  PROC DrawPart154()
    MoveL Offs(pOrigin,203.09,148.13,0.00),v40,z0,tPen\WObj:=wPaper;
    MoveL Offs(pOrigin,201.29,146.33,0.00),v40,z0,tPen\WObj:=wPaper;
    MoveL Offs(pOrigin,200.72,146.00,0.00),v40,z0,tPen\WObj:=wPaper;
    MoveL Offs(pOrigin,205.53,141.19,0.00),v40,z0,tPen\WObj:=wPaper;
    MoveL Offs(pOrigin,205.02,141.09,0.00),v40,z0,tPen\WObj:=wPaper;
    MoveL Offs(pOrigin,203.22,139.29,0.00),v40,z0,tPen\WObj:=wPaper;
    MoveL Offs(pOrigin,203.68,139.61,0.00),v40,z0,tPen\WObj:=wPaper;
    MoveL Offs(pOrigin,204.95,139.61,0.00),v40,z0,tPen\WObj:=wPaper;
    MoveL Offs(pOrigin,205.31,139.90,0.00),v40,z0,tPen\WObj:=wPaper;
    MoveL Offs(pOrigin,203.51,138.09,0.00),v40,z0,tPen\WObj:=wPaper;
    MoveL Offs(pOrigin,202.84,137.91,0.00),v40,z0,tPen\WObj:=wPaper;
    MoveL Offs(pOrigin,207.80,132.95,0.00),v40,z0,tPen\WObj:=wPaper;
    MoveL Offs(pOrigin,207.24,132.86,0.00),v40,z0,tPen\WObj:=wPaper;
    MoveL Offs(pOrigin,205.44,131.06,0.00),v40,z0,tPen\WObj:=wPaper;
    MoveL Offs(pOrigin,206.01,131.16,0.00),v40,z0,tPen\WObj:=wPaper;
    MoveL Offs(pOrigin,207.29,131.16,0.00),v40,z0,tPen\WObj:=wPaper;
    MoveL Offs(pOrigin,207.69,131.82,0.00),v40,z0,tPen\WObj:=wPaper;
    MoveL Offs(pOrigin,205.73,129.86,0.00),v40,z0,tPen\WObj:=wPaper;
    MoveL Offs(pOrigin,206.23,130.10,0.00),v40,z0,tPen\WObj:=wPaper;
    MoveL Offs(pOrigin,207.71,130.10,0.00),v40,z0,tPen\WObj:=wPaper;
    MoveL Offs(pOrigin,208.13,130.77,0.00),v40,z0,tPen\WObj:=wPaper;
    MoveL Offs(pOrigin,205.88,128.51,0.00),v40,z0,tPen\WObj:=wPaper;
    MoveL Offs(pOrigin,206.44,129.05,0.00),v40,z0,tPen\WObj:=wPaper;
    MoveL Offs(pOrigin,207.92,129.05,0.00),v40,z0,tPen\WObj:=wPaper;
    MoveL Offs(pOrigin,208.28,129.42,0.00),v40,z0,tPen\WObj:=wPaper;
    MoveL Offs(pOrigin,206.02,127.17,0.00),v40,z0,tPen\WObj:=wPaper;
    MoveL Offs(pOrigin,206.86,126.94,0.00),v40,z0,tPen\WObj:=wPaper;
    MoveL Offs(pOrigin,208.56,126.94,0.00),v40,z0,tPen\WObj:=wPaper;
    MoveL Offs(pOrigin,209.02,127.18,0.00),v40,z0,tPen\WObj:=wPaper;
    MoveL Offs(pOrigin,206.47,124.62,0.00),v40,z0,tPen\WObj:=wPaper;
    MoveL Offs(pOrigin,206.03,124.27,0.00),v40,z0,tPen\WObj:=wPaper;
    MoveL Offs(pOrigin,212.04,118.26,0.00),v40,z0,tPen\WObj:=wPaper;
    MoveL Offs(pOrigin,211.69,117.90,0.00),v40,z0,tPen\WObj:=wPaper;
    MoveL Offs(pOrigin,208.23,114.44,0.00),v40,z0,tPen\WObj:=wPaper;
    MoveL Offs(pOrigin,207.56,113.77,0.00),v40,z0,tPen\WObj:=wPaper;
    MoveL Offs(pOrigin,215.37,105.96,0.00),v40,z0,tPen\WObj:=wPaper;
    MoveL Offs(pOrigin,214.65,105.92,0.00),v40,z0,tPen\WObj:=wPaper;
    MoveL Offs(pOrigin,212.99,104.27,0.00),v40,z0,tPen\WObj:=wPaper;
    MoveL Offs(pOrigin,213.24,104.76,0.00),v40,z0,tPen\WObj:=wPaper;
    MoveL Offs(pOrigin,214.51,104.76,0.00),v40,z0,tPen\WObj:=wPaper;
    MoveL Offs(pOrigin,215.09,104.87,0.00),v40,z0,tPen\WObj:=wPaper;
    MoveL Offs(pOrigin,213.14,102.92,0.00),v40,z0,tPen\WObj:=wPaper;
    MoveL Offs(pOrigin,212.53,102.82,0.00),v40,z0,tPen\WObj:=wPaper;
    MoveL Offs(pOrigin,216.89,98.47,0.00),v40,z0,tPen\WObj:=wPaper;
    MoveL Offs(pOrigin,216.42,98.74,0.00),v40,z0,tPen\WObj:=wPaper;
    MoveL Offs(pOrigin,214.47,96.78,0.00),v40,z0,tPen\WObj:=wPaper;
    MoveL Offs(pOrigin,214.72,97.37,0.00),v40,z0,tPen\WObj:=wPaper;
    MoveL Offs(pOrigin,216.00,97.37,0.00),v40,z0,tPen\WObj:=wPaper;
    MoveL Offs(pOrigin,216.57,97.39,0.00),v40,z0,tPen\WObj:=wPaper;
    MoveL Offs(pOrigin,214.47,95.29,0.00),v40,z0,tPen\WObj:=wPaper;
    MoveL Offs(pOrigin,214.06,95.33,0.00),v40,z0,tPen\WObj:=wPaper;
    MoveL Offs(pOrigin,217.96,91.42,0.00),v40,z0,tPen\WObj:=wPaper;
    MoveL Offs(pOrigin,217.45,90.80,0.00),v40,z0,tPen\WObj:=wPaper;
    MoveL Offs(pOrigin,215.49,88.85,0.00),v40,z0,tPen\WObj:=wPaper;
    MoveL Offs(pOrigin,216.00,88.92,0.00),v40,z0,tPen\WObj:=wPaper;
    MoveL Offs(pOrigin,217.28,88.92,0.00),v40,z0,tPen\WObj:=wPaper;
    MoveL Offs(pOrigin,217.59,89.45,0.00),v40,z0,tPen\WObj:=wPaper;
    MoveL Offs(pOrigin,215.49,87.35,0.00),v40,z0,tPen\WObj:=wPaper;
    MoveL Offs(pOrigin,215.13,86.79,0.00),v40,z0,tPen\WObj:=wPaper;
    MoveL Offs(pOrigin,218.74,83.18,0.00),v40,z0,tPen\WObj:=wPaper;
    MoveL Offs(pOrigin,218.17,82.56,0.00),v40,z0,tPen\WObj:=wPaper;
    MoveL Offs(pOrigin,216.07,80.46,0.00),v40,z0,tPen\WObj:=wPaper;
    MoveL Offs(pOrigin,216.64,80.47,0.00),v40,z0,tPen\WObj:=wPaper;
    MoveL Offs(pOrigin,217.91,80.47,0.00),v40,z0,tPen\WObj:=wPaper;
    MoveL Offs(pOrigin,218.17,81.07,0.00),v40,z0,tPen\WObj:=wPaper;
    MoveL Offs(pOrigin,216.06,78.96,0.00),v40,z0,tPen\WObj:=wPaper;
    MoveL Offs(pOrigin,215.60,78.85,0.00),v40,z0,tPen\WObj:=wPaper;
    MoveL Offs(pOrigin,218.91,75.54,0.00),v40,z0,tPen\WObj:=wPaper;
    MoveL Offs(pOrigin,218.45,75.37,0.00),v40,z0,tPen\WObj:=wPaper;
    MoveL Offs(pOrigin,216.04,72.97,0.00),v40,z0,tPen\WObj:=wPaper;
    MoveL Offs(pOrigin,215.62,72.85,0.00),v40,z0,tPen\WObj:=wPaper;
    MoveL Offs(pOrigin,218.93,69.55,0.00),v40,z0,tPen\WObj:=wPaper;
    MoveL Offs(pOrigin,218.58,69.53,0.00),v40,z0,tPen\WObj:=wPaper;
    MoveL Offs(pOrigin,211.67,62.62,0.00),v40,z0,tPen\WObj:=wPaper;
    MoveL Offs(pOrigin,211.54,62.80,0.00),v40,z0,tPen\WObj:=wPaper;
    MoveL Offs(pOrigin,211.11,63.22,0.00),v40,z0,tPen\WObj:=wPaper;
    MoveL Offs(pOrigin,211.54,62.80,0.00),v40,fine,tPen\WObj:=wPaper;
    MoveL Offs(pOrigin,211.54,62.80,6.00),v60,z5,tPen\WObj:=wPaper;
    MoveL Offs(pOrigin,212.26,61.72,6.00),vTravel,z5,tPen\WObj:=wPaper;
    MoveL Offs(pOrigin,212.26,61.72,0.00),v60,z0,tPen\WObj:=wPaper;
    MoveL Offs(pOrigin,218.28,67.73,0.00),v40,z0,tPen\WObj:=wPaper;
    MoveL Offs(pOrigin,217.91,67.80,0.00),v40,z0,tPen\WObj:=wPaper;
    MoveL Offs(pOrigin,214.51,67.80,0.00),v40,z0,tPen\WObj:=wPaper;
    MoveL Offs(pOrigin,214.08,68.02,0.00),v40,z0,tPen\WObj:=wPaper;
    MoveL Offs(pOrigin,218.59,72.53,0.00),v40,z0,tPen\WObj:=wPaper;
    MoveL Offs(pOrigin,218.92,72.55,0.00),v40,z0,tPen\WObj:=wPaper;
    MoveL Offs(pOrigin,215.61,75.85,0.00),v40,z0,tPen\WObj:=wPaper;
    MoveL Offs(pOrigin,216.05,75.97,0.00),v40,z0,tPen\WObj:=wPaper;
    MoveL Offs(pOrigin,218.46,78.37,0.00),v40,z0,tPen\WObj:=wPaper;
    MoveL Offs(pOrigin,218.90,78.54,0.00),v40,z0,tPen\WObj:=wPaper;
    MoveL Offs(pOrigin,215.44,81.99,0.00),v40,z0,tPen\WObj:=wPaper;
    MoveL Offs(pOrigin,215.92,81.81,0.00),v40,z0,tPen\WObj:=wPaper;
    MoveL Offs(pOrigin,218.03,83.91,0.00),v40,z0,tPen\WObj:=wPaper;
    MoveL Offs(pOrigin,217.70,83.64,0.00),v40,z0,tPen\WObj:=wPaper;
    MoveL Offs(pOrigin,216.42,83.64,0.00),v40,z0,tPen\WObj:=wPaper;
    MoveL Offs(pOrigin,215.93,83.31,0.00),v40,z0,tPen\WObj:=wPaper;
    MoveL Offs(pOrigin,218.03,85.41,0.00),v40,z0,tPen\WObj:=wPaper;
    MoveL Offs(pOrigin,217.49,85.75,0.00),v40,z0,tPen\WObj:=wPaper;
    MoveL Offs(pOrigin,216.21,85.75,0.00),v40,z0,tPen\WObj:=wPaper;
    MoveL Offs(pOrigin,215.63,86.00,0.00),v40,z0,tPen\WObj:=wPaper;
    MoveL Offs(pOrigin,217.89,88.26,0.00),v40,z0,tPen\WObj:=wPaper;
    MoveL Offs(pOrigin,218.27,88.13,0.00),v40,z0,tPen\WObj:=wPaper;
    MoveL Offs(pOrigin,214.67,91.73,0.00),v40,z0,tPen\WObj:=wPaper;
    MoveL Offs(pOrigin,215.05,91.39,0.00),v40,z0,tPen\WObj:=wPaper;
    MoveL Offs(pOrigin,217.16,93.50,0.00),v40,z0,tPen\WObj:=wPaper;
    MoveL Offs(pOrigin,217.66,93.22,0.00),v40,z0,tPen\WObj:=wPaper;
    MoveL Offs(pOrigin,213.75,97.13,0.00),v40,z0,tPen\WObj:=wPaper;
    MoveL Offs(pOrigin,214.02,97.83,0.00),v40,z0,tPen\WObj:=wPaper;
    MoveL Offs(pOrigin,216.13,99.93,0.00),v40,z0,tPen\WObj:=wPaper;
    MoveL Offs(pOrigin,216.44,100.42,0.00),v40,z0,tPen\WObj:=wPaper;
    MoveL Offs(pOrigin,212.08,104.77,0.00),v40,z0,tPen\WObj:=wPaper;
    MoveL Offs(pOrigin,212.55,105.32,0.00),v40,z0,tPen\WObj:=wPaper;
    MoveL Offs(pOrigin,214.50,107.27,0.00),v40,z0,tPen\WObj:=wPaper;
    MoveL Offs(pOrigin,214.09,106.87,0.00),v40,z0,tPen\WObj:=wPaper;
    MoveL Offs(pOrigin,212.81,106.87,0.00),v40,z0,tPen\WObj:=wPaper;
    MoveL Offs(pOrigin,212.25,106.51,0.00),v40,z0,tPen\WObj:=wPaper;
    MoveL Offs(pOrigin,214.36,108.62,0.00),v40,z0,tPen\WObj:=wPaper;
    MoveL Offs(pOrigin,214.61,108.21,0.00),v40,z0,tPen\WObj:=wPaper;
    MoveL Offs(pOrigin,207.40,115.42,0.00),v40,z0,tPen\WObj:=wPaper;
    MoveL Offs(pOrigin,207.94,115.64,0.00),v40,z0,tPen\WObj:=wPaper;
  ENDPROC

  PROC DrawPart155()
    MoveL Offs(pOrigin,211.24,118.94,0.00),v40,z0,tPen\WObj:=wPaper;
    MoveL Offs(pOrigin,210.90,118.49,0.00),v40,z0,tPen\WObj:=wPaper;
    MoveL Offs(pOrigin,209.41,118.49,0.00),v40,z0,tPen\WObj:=wPaper;
    MoveL Offs(pOrigin,209.84,117.43,0.00),v40,z0,tPen\WObj:=wPaper;
    MoveL Offs(pOrigin,211.32,117.43,0.00),v40,z0,tPen\WObj:=wPaper;
    MoveL Offs(pOrigin,211.98,116.70,0.00),v40,z0,tPen\WObj:=wPaper;
    MoveL Offs(pOrigin,208.53,113.24,0.00),v40,fine,tPen\WObj:=wPaper;
    MoveL Offs(pOrigin,208.53,113.24,6.00),v60,z5,tPen\WObj:=wPaper;
    MoveL Offs(pOrigin,207.86,111.98,6.00),vTravel,z5,tPen\WObj:=wPaper;
    MoveL Offs(pOrigin,207.86,111.98,0.00),v60,z0,tPen\WObj:=wPaper;
    MoveL Offs(pOrigin,210.27,109.57,0.00),v40,z0,tPen\WObj:=wPaper;
    MoveL Offs(pOrigin,211.02,108.82,0.00),v40,z0,tPen\WObj:=wPaper;
    MoveL Offs(pOrigin,215.83,104.01,0.00),v40,z0,tPen\WObj:=wPaper;
    MoveL Offs(pOrigin,215.39,103.68,0.00),v40,z0,tPen\WObj:=wPaper;
    MoveL Offs(pOrigin,213.44,101.72,0.00),v40,z0,tPen\WObj:=wPaper;
    MoveL Offs(pOrigin,214.09,101.59,0.00),v40,z0,tPen\WObj:=wPaper;
    MoveL Offs(pOrigin,215.15,101.59,0.00),v40,z0,tPen\WObj:=wPaper;
    MoveL Offs(pOrigin,215.83,101.13,0.00),v40,z0,tPen\WObj:=wPaper;
    MoveL Offs(pOrigin,213.88,99.18,0.00),v40,z0,tPen\WObj:=wPaper;
    MoveL Offs(pOrigin,213.45,98.93,0.00),v40,z0,tPen\WObj:=wPaper;
    MoveL Offs(pOrigin,217.50,94.87,0.00),v40,z0,tPen\WObj:=wPaper;
    MoveL Offs(pOrigin,217.01,94.84,0.00),v40,z0,tPen\WObj:=wPaper;
    MoveL Offs(pOrigin,214.76,92.59,0.00),v40,z0,tPen\WObj:=wPaper;
    MoveL Offs(pOrigin,215.58,92.09,0.00),v40,z0,tPen\WObj:=wPaper;
    MoveL Offs(pOrigin,216.85,92.09,0.00),v40,z0,tPen\WObj:=wPaper;
    MoveL Offs(pOrigin,217.15,92.00,0.00),v40,z0,tPen\WObj:=wPaper;
    MoveL Offs(pOrigin,215.20,90.04,0.00),v40,z0,tPen\WObj:=wPaper;
    MoveL Offs(pOrigin,214.82,90.08,0.00),v40,z0,tPen\WObj:=wPaper;
    MoveL Offs(pOrigin,218.58,86.33,0.00),v40,z0,tPen\WObj:=wPaper;
    MoveL Offs(pOrigin,217.88,86.76,0.00),v40,z0,tPen\WObj:=wPaper;
    MoveL Offs(pOrigin,215.63,84.50,0.00),v40,z0,tPen\WObj:=wPaper;
    MoveL Offs(pOrigin,215.28,85.14,0.00),v40,z0,tPen\WObj:=wPaper;
    MoveL Offs(pOrigin,218.74,81.68,0.00),v40,z0,tPen\WObj:=wPaper;
    MoveL Offs(pOrigin,217.91,81.53,0.00),v40,z0,tPen\WObj:=wPaper;
    MoveL Offs(pOrigin,216.64,81.53,0.00),v40,z0,tPen\WObj:=wPaper;
    MoveL Offs(pOrigin,216.64,82.58,0.00),v40,z0,tPen\WObj:=wPaper;
    MoveL Offs(pOrigin,217.70,82.58,0.00),v40,fine,tPen\WObj:=wPaper;
    MoveL Offs(pOrigin,217.70,82.58,6.00),v60,z5,tPen\WObj:=wPaper;
    MoveL Offs(pOrigin,217.49,84.70,6.00),vTravel,z5,tPen\WObj:=wPaper;
    MoveL Offs(pOrigin,217.49,84.70,0.00),v60,z0,tPen\WObj:=wPaper;
    MoveL Offs(pOrigin,216.42,84.70,0.00),v40,fine,tPen\WObj:=wPaper;
    MoveL Offs(pOrigin,216.42,84.70,6.00),v60,z5,tPen\WObj:=wPaper;
    MoveL Offs(pOrigin,215.29,83.64,6.00),vTravel,z5,tPen\WObj:=wPaper;
    MoveL Offs(pOrigin,215.29,83.64,0.00),v60,z0,tPen\WObj:=wPaper;
    MoveL Offs(pOrigin,219.05,79.88,0.00),v40,z0,tPen\WObj:=wPaper;
    MoveL Offs(pOrigin,218.46,79.87,0.00),v40,z0,tPen\WObj:=wPaper;
    MoveL Offs(pOrigin,216.06,77.46,0.00),v40,z0,tPen\WObj:=wPaper;
    MoveL Offs(pOrigin,215.61,77.35,0.00),v40,z0,tPen\WObj:=wPaper;
    MoveL Offs(pOrigin,218.91,74.04,0.00),v40,z0,tPen\WObj:=wPaper;
    MoveL Offs(pOrigin,218.59,74.03,0.00),v40,z0,tPen\WObj:=wPaper;
    MoveL Offs(pOrigin,213.79,69.22,0.00),v40,z0,tPen\WObj:=wPaper;
    MoveL Offs(pOrigin,214.09,69.91,0.00),v40,z0,tPen\WObj:=wPaper;
    MoveL Offs(pOrigin,217.91,69.91,0.00),v40,z0,tPen\WObj:=wPaper;
    MoveL Offs(pOrigin,217.91,68.86,0.00),v40,z0,tPen\WObj:=wPaper;
    MoveL Offs(pOrigin,214.51,68.86,0.00),v40,z0,tPen\WObj:=wPaper;
    MoveL Offs(pOrigin,215.44,68.54,0.00),v40,z0,tPen\WObj:=wPaper;
    MoveL Offs(pOrigin,215.44,59.82,0.00),v40,fine,tPen\WObj:=wPaper;
    MoveL Offs(pOrigin,215.44,59.82,6.00),v60,z5,tPen\WObj:=wPaper;
    MoveL Offs(pOrigin,213.76,60.23,6.00),vTravel,z5,tPen\WObj:=wPaper;
    MoveL Offs(pOrigin,213.76,60.23,0.00),v60,z0,tPen\WObj:=wPaper;
    MoveL Offs(pOrigin,218.12,64.59,0.00),v40,z0,tPen\WObj:=wPaper;
    MoveL Offs(pOrigin,217.49,64.63,0.00),v40,z0,tPen\WObj:=wPaper;
    MoveL Offs(pOrigin,214.51,64.63,0.00),v40,z0,tPen\WObj:=wPaper;
    MoveL Offs(pOrigin,214.51,65.69,0.00),v40,z0,tPen\WObj:=wPaper;
    MoveL Offs(pOrigin,217.70,65.69,0.00),v40,z0,tPen\WObj:=wPaper;
    MoveL Offs(pOrigin,217.70,66.74,0.00),v40,z0,tPen\WObj:=wPaper;
    MoveL Offs(pOrigin,214.51,66.74,0.00),v40,z0,tPen\WObj:=wPaper;
    MoveL Offs(pOrigin,214.08,66.52,0.00),v40,z0,tPen\WObj:=wPaper;
    MoveL Offs(pOrigin,218.59,71.03,0.00),v40,z0,tPen\WObj:=wPaper;
    MoveL Offs(pOrigin,218.92,71.05,0.00),v40,z0,tPen\WObj:=wPaper;
    MoveL Offs(pOrigin,215.62,74.35,0.00),v40,z0,tPen\WObj:=wPaper;
    MoveL Offs(pOrigin,216.05,74.47,0.00),v40,z0,tPen\WObj:=wPaper;
    MoveL Offs(pOrigin,218.45,76.87,0.00),v40,z0,tPen\WObj:=wPaper;
    MoveL Offs(pOrigin,218.90,77.04,0.00),v40,z0,tPen\WObj:=wPaper;
    MoveL Offs(pOrigin,215.45,80.50,0.00),v40,fine,tPen\WObj:=wPaper;
    MoveL Offs(pOrigin,215.45,80.50,6.00),v60,z5,tPen\WObj:=wPaper;
    MoveL Offs(pOrigin,216.64,79.42,6.00),vTravel,z5,tPen\WObj:=wPaper;
    MoveL Offs(pOrigin,216.64,79.42,0.00),v60,z0,tPen\WObj:=wPaper;
    MoveL Offs(pOrigin,217.91,79.42,0.00),v40,z0,tPen\WObj:=wPaper;
    MoveL Offs(pOrigin,217.91,78.36,0.00),v40,z0,tPen\WObj:=wPaper;
    MoveL Offs(pOrigin,216.85,78.36,0.00),v40,z0,tPen\WObj:=wPaper;
    MoveL Offs(pOrigin,216.85,77.30,0.00),v40,z0,tPen\WObj:=wPaper;
    MoveL Offs(pOrigin,217.91,77.30,0.00),v40,z0,tPen\WObj:=wPaper;
    MoveL Offs(pOrigin,217.91,76.25,0.00),v40,z0,tPen\WObj:=wPaper;
    MoveL Offs(pOrigin,216.85,76.25,0.00),v40,z0,tPen\WObj:=wPaper;
    MoveL Offs(pOrigin,216.85,75.19,0.00),v40,z0,tPen\WObj:=wPaper;
    MoveL Offs(pOrigin,217.91,75.19,0.00),v40,z0,tPen\WObj:=wPaper;
    MoveL Offs(pOrigin,217.91,74.14,0.00),v40,z0,tPen\WObj:=wPaper;
    MoveL Offs(pOrigin,216.85,74.14,0.00),v40,z0,tPen\WObj:=wPaper;
    MoveL Offs(pOrigin,216.85,73.08,0.00),v40,z0,tPen\WObj:=wPaper;
    MoveL Offs(pOrigin,217.91,73.08,0.00),v40,z0,tPen\WObj:=wPaper;
    MoveL Offs(pOrigin,217.91,72.02,0.00),v40,z0,tPen\WObj:=wPaper;
    MoveL Offs(pOrigin,216.85,72.02,0.00),v40,z0,tPen\WObj:=wPaper;
    MoveL Offs(pOrigin,216.85,70.97,0.00),v40,z0,tPen\WObj:=wPaper;
    MoveL Offs(pOrigin,217.91,70.97,0.00),v40,fine,tPen\WObj:=wPaper;
    MoveL Offs(pOrigin,217.91,70.97,6.00),v60,z5,tPen\WObj:=wPaper;
    MoveL Offs(pOrigin,218.63,68.35,6.00),vTravel,z5,tPen\WObj:=wPaper;
    MoveL Offs(pOrigin,218.63,68.35,0.00),v60,z0,tPen\WObj:=wPaper;
    MoveL Offs(pOrigin,212.77,74.21,0.00),v40,z0,tPen\WObj:=wPaper;
    MoveL Offs(pOrigin,212.60,74.01,0.00),v40,z0,tPen\WObj:=wPaper;
    MoveL Offs(pOrigin,210.95,72.36,0.00),v40,z0,tPen\WObj:=wPaper;
    MoveL Offs(pOrigin,210.26,73.08,0.00),v40,z0,tPen\WObj:=wPaper;
    MoveL Offs(pOrigin,212.60,73.08,0.00),v40,z0,tPen\WObj:=wPaper;
    MoveL Offs(pOrigin,213.24,73.00,0.00),v40,z0,tPen\WObj:=wPaper;
    MoveL Offs(pOrigin,213.52,72.86,0.00),v40,z0,tPen\WObj:=wPaper;
    MoveL Offs(pOrigin,210.90,74.35,0.00),v40,z0,tPen\WObj:=wPaper;
    MoveL Offs(pOrigin,206.86,75.55,0.00),v40,z0,tPen\WObj:=wPaper;
    MoveL Offs(pOrigin,204.10,75.97,0.00),v40,z0,tPen\WObj:=wPaper;
    MoveL Offs(pOrigin,194.96,76.47,0.00),v40,z0,tPen\WObj:=wPaper;
    MoveL Offs(pOrigin,190.50,80.22,0.00),v40,z0,tPen\WObj:=wPaper;
    MoveL Offs(pOrigin,189.86,81.93,0.00),v40,z0,tPen\WObj:=wPaper;
    MoveL Offs(pOrigin,187.74,84.05,0.00),v40,z0,tPen\WObj:=wPaper;
    MoveL Offs(pOrigin,178.03,92.34,0.00),v40,z0,tPen\WObj:=wPaper;
    MoveL Offs(pOrigin,182.14,100.20,0.00),v40,z0,tPen\WObj:=wPaper;
    MoveL Offs(pOrigin,187.74,108.06,0.00),v40,z0,tPen\WObj:=wPaper;
    MoveL Offs(pOrigin,193.26,113.80,0.00),v40,z0,tPen\WObj:=wPaper;
    MoveL Offs(pOrigin,196.24,116.35,0.00),v40,z0,tPen\WObj:=wPaper;
    MoveL Offs(pOrigin,199.64,118.69,0.00),v40,fine,tPen\WObj:=wPaper;
    MoveL Offs(pOrigin,199.64,118.69,6.00),v60,z5,tPen\WObj:=wPaper;
    MoveL Offs(pOrigin,206.94,118.87,6.00),vTravel,z5,tPen\WObj:=wPaper;
  ENDPROC

  PROC DrawPart156()
    MoveL Offs(pOrigin,206.94,118.87,0.00),v60,z0,tPen\WObj:=wPaper;
    MoveL Offs(pOrigin,213.55,112.26,0.00),v40,z0,tPen\WObj:=wPaper;
    MoveL Offs(pOrigin,213.32,112.06,0.00),v40,z0,tPen\WObj:=wPaper;
    MoveL Offs(pOrigin,211.52,110.26,0.00),v40,z0,tPen\WObj:=wPaper;
    MoveL Offs(pOrigin,211.96,110.04,0.00),v40,z0,tPen\WObj:=wPaper;
    MoveL Offs(pOrigin,213.24,110.04,0.00),v40,z0,tPen\WObj:=wPaper;
    MoveL Offs(pOrigin,213.91,109.66,0.00),v40,z0,tPen\WObj:=wPaper;
    MoveL Offs(pOrigin,212.11,107.86,0.00),v40,z0,tPen\WObj:=wPaper;
    MoveL Offs(pOrigin,212.60,107.93,0.00),v40,z0,tPen\WObj:=wPaper;
    MoveL Offs(pOrigin,213.66,107.93,0.00),v40,z0,tPen\WObj:=wPaper;
    MoveL Offs(pOrigin,213.45,108.98,0.00),v40,z0,tPen\WObj:=wPaper;
    MoveL Offs(pOrigin,212.18,108.98,0.00),v40,z0,tPen\WObj:=wPaper;
    MoveL Offs(pOrigin,211.66,108.91,0.00),v40,z0,tPen\WObj:=wPaper;
    MoveL Offs(pOrigin,213.61,110.86,0.00),v40,z0,tPen\WObj:=wPaper;
    MoveL Offs(pOrigin,212.81,111.10,0.00),v40,z0,tPen\WObj:=wPaper;
    MoveL Offs(pOrigin,211.75,111.10,0.00),v40,z0,tPen\WObj:=wPaper;
    MoveL Offs(pOrigin,211.07,111.30,0.00),v40,z0,tPen\WObj:=wPaper;
    MoveL Offs(pOrigin,213.02,113.26,0.00),v40,z0,tPen\WObj:=wPaper;
    MoveL Offs(pOrigin,212.39,113.21,0.00),v40,z0,tPen\WObj:=wPaper;
    MoveL Offs(pOrigin,211.11,113.21,0.00),v40,z0,tPen\WObj:=wPaper;
    MoveL Offs(pOrigin,210.77,112.50,0.00),v40,z0,tPen\WObj:=wPaper;
    MoveL Offs(pOrigin,212.58,114.30,0.00),v40,z0,tPen\WObj:=wPaper;
    MoveL Offs(pOrigin,211.96,114.26,0.00),v40,z0,tPen\WObj:=wPaper;
    MoveL Offs(pOrigin,210.90,114.26,0.00),v40,z0,tPen\WObj:=wPaper;
    MoveL Offs(pOrigin,210.33,113.55,0.00),v40,z0,tPen\WObj:=wPaper;
    MoveL Offs(pOrigin,212.28,115.50,0.00),v40,z0,tPen\WObj:=wPaper;
    MoveL Offs(pOrigin,211.75,115.32,0.00),v40,z0,tPen\WObj:=wPaper;
    MoveL Offs(pOrigin,210.48,115.32,0.00),v40,z0,tPen\WObj:=wPaper;
    MoveL Offs(pOrigin,210.05,116.38,0.00),v40,z0,tPen\WObj:=wPaper;
    MoveL Offs(pOrigin,211.54,116.38,0.00),v40,z0,tPen\WObj:=wPaper;
    MoveL Offs(pOrigin,212.49,116.31,0.00),v40,z0,tPen\WObj:=wPaper;
    MoveL Offs(pOrigin,206.48,122.32,0.00),v40,z0,tPen\WObj:=wPaper;
    MoveL Offs(pOrigin,207.06,122.23,0.00),v40,z0,tPen\WObj:=wPaper;
    MoveL Offs(pOrigin,209.61,124.78,0.00),v40,z0,tPen\WObj:=wPaper;
    MoveL Offs(pOrigin,209.20,124.82,0.00),v40,z0,tPen\WObj:=wPaper;
    MoveL Offs(pOrigin,207.08,124.82,0.00),v40,z0,tPen\WObj:=wPaper;
    MoveL Offs(pOrigin,206.86,125.88,0.00),v40,z0,tPen\WObj:=wPaper;
    MoveL Offs(pOrigin,208.99,125.88,0.00),v40,z0,tPen\WObj:=wPaper;
    MoveL Offs(pOrigin,209.32,125.98,0.00),v40,z0,tPen\WObj:=wPaper;
    MoveL Offs(pOrigin,206.76,123.42,0.00),v40,z0,tPen\WObj:=wPaper;
    MoveL Offs(pOrigin,207.50,123.77,0.00),v40,z0,tPen\WObj:=wPaper;
    MoveL Offs(pOrigin,209.41,123.77,0.00),v40,z0,tPen\WObj:=wPaper;
    MoveL Offs(pOrigin,209.91,123.58,0.00),v40,z0,tPen\WObj:=wPaper;
    MoveL Offs(pOrigin,207.35,121.03,0.00),v40,z0,tPen\WObj:=wPaper;
    MoveL Offs(pOrigin,206.79,120.52,0.00),v40,z0,tPen\WObj:=wPaper;
    MoveL Offs(pOrigin,213.25,114.06,0.00),v40,fine,tPen\WObj:=wPaper;
    MoveL Offs(pOrigin,213.25,114.06,6.00),v60,z5,tPen\WObj:=wPaper;
    MoveL Offs(pOrigin,212.60,112.15,6.00),vTravel,z5,tPen\WObj:=wPaper;
    MoveL Offs(pOrigin,212.60,112.15,0.00),v60,z0,tPen\WObj:=wPaper;
    MoveL Offs(pOrigin,211.54,112.15,0.00),v40,fine,tPen\WObj:=wPaper;
    MoveL Offs(pOrigin,211.54,112.15,6.00),v60,z5,tPen\WObj:=wPaper;
    MoveL Offs(pOrigin,214.31,110.01,6.00),vTravel,z5,tPen\WObj:=wPaper;
    MoveL Offs(pOrigin,214.31,110.01,0.00),v60,z0,tPen\WObj:=wPaper;
    MoveL Offs(pOrigin,207.25,117.07,0.00),v40,z0,tPen\WObj:=wPaper;
    MoveL Offs(pOrigin,207.79,116.99,0.00),v40,z0,tPen\WObj:=wPaper;
    MoveL Offs(pOrigin,210.95,120.14,0.00),v40,z0,tPen\WObj:=wPaper;
    MoveL Offs(pOrigin,211.43,120.35,0.00),v40,z0,tPen\WObj:=wPaper;
    MoveL Offs(pOrigin,205.87,125.91,0.00),v40,z0,tPen\WObj:=wPaper;
    MoveL Offs(pOrigin,206.32,125.97,0.00),v40,z0,tPen\WObj:=wPaper;
    MoveL Offs(pOrigin,208.72,128.37,0.00),v40,z0,tPen\WObj:=wPaper;
    MoveL Offs(pOrigin,209.16,128.60,0.00),v40,z0,tPen\WObj:=wPaper;
    MoveL Offs(pOrigin,204.20,133.56,0.00),v40,z0,tPen\WObj:=wPaper;
    MoveL Offs(pOrigin,204.85,133.45,0.00),v40,z0,tPen\WObj:=wPaper;
    MoveL Offs(pOrigin,206.65,135.26,0.00),v40,z0,tPen\WObj:=wPaper;
    MoveL Offs(pOrigin,206.23,135.38,0.00),v40,z0,tPen\WObj:=wPaper;
    MoveL Offs(pOrigin,204.95,135.38,0.00),v40,z0,tPen\WObj:=wPaper;
    MoveL Offs(pOrigin,204.25,135.85,0.00),v40,z0,tPen\WObj:=wPaper;
    MoveL Offs(pOrigin,205.91,137.50,0.00),v40,z0,tPen\WObj:=wPaper;
    MoveL Offs(pOrigin,205.59,137.50,0.00),v40,z0,tPen\WObj:=wPaper;
    MoveL Offs(pOrigin,204.31,137.50,0.00),v40,z0,tPen\WObj:=wPaper;
    MoveL Offs(pOrigin,203.81,136.90,0.00),v40,z0,tPen\WObj:=wPaper;
    MoveL Offs(pOrigin,205.61,138.70,0.00),v40,z0,tPen\WObj:=wPaper;
    MoveL Offs(pOrigin,205.16,138.55,0.00),v40,z0,tPen\WObj:=wPaper;
    MoveL Offs(pOrigin,204.10,138.55,0.00),v40,fine,tPen\WObj:=wPaper;
    MoveL Offs(pOrigin,204.10,138.55,6.00),v60,z5,tPen\WObj:=wPaper;
    MoveL Offs(pOrigin,205.83,139.40,6.00),vTravel,z5,tPen\WObj:=wPaper;
    MoveL Offs(pOrigin,205.83,139.40,0.00),v60,z0,tPen\WObj:=wPaper;
    MoveL Offs(pOrigin,201.32,143.90,0.00),v40,z0,tPen\WObj:=wPaper;
    MoveL Offs(pOrigin,201.88,143.93,0.00),v40,z0,tPen\WObj:=wPaper;
    MoveL Offs(pOrigin,203.68,145.73,0.00),v40,z0,tPen\WObj:=wPaper;
    MoveL Offs(pOrigin,203.04,145.94,0.00),v40,z0,tPen\WObj:=wPaper;
    MoveL Offs(pOrigin,201.98,145.94,0.00),v40,z0,tPen\WObj:=wPaper;
    MoveL Offs(pOrigin,201.74,145.28,0.00),v40,z0,tPen\WObj:=wPaper;
    MoveL Offs(pOrigin,203.39,146.93,0.00),v40,z0,tPen\WObj:=wPaper;
    MoveL Offs(pOrigin,202.82,147.00,0.00),v40,z0,tPen\WObj:=wPaper;
    MoveL Offs(pOrigin,201.76,147.00,0.00),v40,fine,tPen\WObj:=wPaper;
    MoveL Offs(pOrigin,201.76,147.00,6.00),v60,z5,tPen\WObj:=wPaper;
    MoveL Offs(pOrigin,200.41,147.80,6.00),vTravel,z5,tPen\WObj:=wPaper;
    MoveL Offs(pOrigin,200.41,147.80,0.00),v60,z0,tPen\WObj:=wPaper;
    MoveL Offs(pOrigin,205.22,142.99,0.00),v40,z0,tPen\WObj:=wPaper;
    MoveL Offs(pOrigin,204.72,142.29,0.00),v40,z0,tPen\WObj:=wPaper;
    MoveL Offs(pOrigin,202.92,140.49,0.00),v40,z0,tPen\WObj:=wPaper;
    MoveL Offs(pOrigin,203.46,140.66,0.00),v40,z0,tPen\WObj:=wPaper;
    MoveL Offs(pOrigin,204.52,140.66,0.00),v40,z0,tPen\WObj:=wPaper;
    MoveL Offs(pOrigin,204.31,141.72,0.00),v40,z0,tPen\WObj:=wPaper;
    MoveL Offs(pOrigin,203.25,141.72,0.00),v40,z0,tPen\WObj:=wPaper;
    MoveL Offs(pOrigin,202.47,141.54,0.00),v40,z0,tPen\WObj:=wPaper;
    MoveL Offs(pOrigin,204.28,143.34,0.00),v40,z0,tPen\WObj:=wPaper;
    MoveL Offs(pOrigin,204.10,142.78,0.00),v40,z0,tPen\WObj:=wPaper;
    MoveL Offs(pOrigin,202.82,142.78,0.00),v40,z0,tPen\WObj:=wPaper;
    MoveL Offs(pOrigin,202.33,142.88,0.00),v40,z0,tPen\WObj:=wPaper;
    MoveL Offs(pOrigin,204.13,144.69,0.00),v40,z0,tPen\WObj:=wPaper;
    MoveL Offs(pOrigin,204.62,145.09,0.00),v40,z0,tPen\WObj:=wPaper;
    MoveL Offs(pOrigin,199.81,149.90,0.00),v40,fine,tPen\WObj:=wPaper;
    MoveL Offs(pOrigin,199.81,149.90,6.00),v60,z5,tPen\WObj:=wPaper;
    MoveL Offs(pOrigin,199.35,151.85,6.00),vTravel,z5,tPen\WObj:=wPaper;
    MoveL Offs(pOrigin,199.35,151.85,0.00),v60,z0,tPen\WObj:=wPaper;
    MoveL Offs(pOrigin,203.86,147.34,0.00),v40,fine,tPen\WObj:=wPaper;
    MoveL Offs(pOrigin,203.86,147.34,6.00),v60,z5,tPen\WObj:=wPaper;
    MoveL Offs(pOrigin,203.25,149.44,6.00),vTravel,z5,tPen\WObj:=wPaper;
    MoveL Offs(pOrigin,203.25,149.44,0.00),v60,z0,tPen\WObj:=wPaper;
    MoveL Offs(pOrigin,198.75,153.95,0.00),v40,z0,tPen\WObj:=wPaper;
    MoveL Offs(pOrigin,199.07,154.56,0.00),v40,z0,tPen\WObj:=wPaper;
    MoveL Offs(pOrigin,200.87,156.36,0.00),v40,z0,tPen\WObj:=wPaper;
    MoveL Offs(pOrigin,200.28,156.50,0.00),v40,z0,tPen\WObj:=wPaper;
    MoveL Offs(pOrigin,199.21,156.50,0.00),v40,z0,tPen\WObj:=wPaper;
    MoveL Offs(pOrigin,198.48,156.95,0.00),v40,z0,tPen\WObj:=wPaper;
    MoveL Offs(pOrigin,200.13,158.61,0.00),v40,z0,tPen\WObj:=wPaper;
    MoveL Offs(pOrigin,200.68,159.48,0.00),v40,z0,tPen\WObj:=wPaper;
    MoveL Offs(pOrigin,196.17,163.99,0.00),v40,z0,tPen\WObj:=wPaper;
  ENDPROC

  PROC DrawPart157()
    MoveL Offs(pOrigin,196.70,164.14,0.00),v40,z0,tPen\WObj:=wPaper;
    MoveL Offs(pOrigin,198.35,165.79,0.00),v40,z0,tPen\WObj:=wPaper;
    MoveL Offs(pOrigin,199.01,165.63,0.00),v40,z0,tPen\WObj:=wPaper;
    MoveL Offs(pOrigin,194.65,169.99,0.00),v40,z0,tPen\WObj:=wPaper;
    MoveL Offs(pOrigin,195.07,169.98,0.00),v40,z0,tPen\WObj:=wPaper;
    MoveL Offs(pOrigin,196.87,171.78,0.00),v40,z0,tPen\WObj:=wPaper;
    MoveL Offs(pOrigin,197.49,171.63,0.00),v40,z0,tPen\WObj:=wPaper;
    MoveL Offs(pOrigin,192.99,176.14,0.00),v40,z0,tPen\WObj:=wPaper;
    MoveL Offs(pOrigin,193.59,175.96,0.00),v40,z0,tPen\WObj:=wPaper;
    MoveL Offs(pOrigin,198.85,181.22,0.00),v40,z0,tPen\WObj:=wPaper;
    MoveL Offs(pOrigin,198.21,181.36,0.00),v40,z0,tPen\WObj:=wPaper;
    MoveL Offs(pOrigin,200.47,179.11,0.00),v40,z0,tPen\WObj:=wPaper;
    MoveL Offs(pOrigin,200.04,179.43,0.00),v40,z0,tPen\WObj:=wPaper;
    MoveL Offs(pOrigin,207.41,186.79,0.00),v40,z0,tPen\WObj:=wPaper;
    MoveL Offs(pOrigin,207.33,187.18,0.00),v40,z0,tPen\WObj:=wPaper;
    MoveL Offs(pOrigin,210.19,184.32,0.00),v40,z0,tPen\WObj:=wPaper;
    MoveL Offs(pOrigin,209.65,184.55,0.00),v40,z0,tPen\WObj:=wPaper;
    MoveL Offs(pOrigin,223.17,198.07,0.00),v40,z0,tPen\WObj:=wPaper;
    MoveL Offs(pOrigin,222.80,197.69,0.00),v40,z0,tPen\WObj:=wPaper;
    MoveL Offs(pOrigin,221.74,197.69,0.00),v40,z0,tPen\WObj:=wPaper;
    MoveL Offs(pOrigin,221.22,197.62,0.00),v40,z0,tPen\WObj:=wPaper;
    MoveL Offs(pOrigin,223.02,199.42,0.00),v40,z0,tPen\WObj:=wPaper;
    MoveL Offs(pOrigin,223.32,199.56,0.00),v40,z0,tPen\WObj:=wPaper;
    MoveL Offs(pOrigin,219.57,203.32,0.00),v40,z0,tPen\WObj:=wPaper;
    MoveL Offs(pOrigin,219.89,203.76,0.00),v40,z0,tPen\WObj:=wPaper;
    MoveL Offs(pOrigin,221.84,205.71,0.00),v40,z0,tPen\WObj:=wPaper;
    MoveL Offs(pOrigin,221.31,205.08,0.00),v40,z0,tPen\WObj:=wPaper;
    MoveL Offs(pOrigin,220.25,205.08,0.00),v40,z0,tPen\WObj:=wPaper;
    MoveL Offs(pOrigin,219.75,205.10,0.00),v40,z0,tPen\WObj:=wPaper;
    MoveL Offs(pOrigin,223.65,209.01,0.00),v40,z0,tPen\WObj:=wPaper;
    MoveL Offs(pOrigin,223.44,208.25,0.00),v40,z0,tPen\WObj:=wPaper;
    MoveL Offs(pOrigin,219.82,208.25,0.00),v40,z0,tPen\WObj:=wPaper;
    MoveL Offs(pOrigin,219.45,207.80,0.00),v40,z0,tPen\WObj:=wPaper;
    MoveL Offs(pOrigin,222.91,211.26,0.00),v40,z0,tPen\WObj:=wPaper;
    MoveL Offs(pOrigin,222.68,212.15,0.00),v40,z0,tPen\WObj:=wPaper;
    MoveL Offs(pOrigin,226.44,208.39,0.00),v40,z0,tPen\WObj:=wPaper;
    MoveL Offs(pOrigin,225.69,207.64,0.00),v40,z0,tPen\WObj:=wPaper;
    MoveL Offs(pOrigin,199.25,234.09,0.00),v40,z0,tPen\WObj:=wPaper;
    MoveL Offs(pOrigin,199.16,233.80,0.00),v40,z0,tPen\WObj:=wPaper;
    MoveL Offs(pOrigin,196.91,231.55,0.00),v40,z0,tPen\WObj:=wPaper;
    MoveL Offs(pOrigin,197.61,231.25,0.00),v40,z0,tPen\WObj:=wPaper;
    MoveL Offs(pOrigin,195.66,233.20,0.00),v40,z0,tPen\WObj:=wPaper;
    MoveL Offs(pOrigin,195.26,232.89,0.00),v40,z0,tPen\WObj:=wPaper;
    MoveL Offs(pOrigin,192.86,230.49,0.00),v40,z0,tPen\WObj:=wPaper;
    MoveL Offs(pOrigin,192.97,229.91,0.00),v40,z0,tPen\WObj:=wPaper;
    MoveL Offs(pOrigin,191.02,231.87,0.00),v40,z0,tPen\WObj:=wPaper;
    MoveL Offs(pOrigin,190.76,231.38,0.00),v40,z0,tPen\WObj:=wPaper;
    MoveL Offs(pOrigin,188.21,228.83,0.00),v40,z0,tPen\WObj:=wPaper;
    MoveL Offs(pOrigin,188.48,228.43,0.00),v40,z0,tPen\WObj:=wPaper;
    MoveL Offs(pOrigin,186.68,230.23,0.00),v40,z0,tPen\WObj:=wPaper;
    MoveL Offs(pOrigin,186.89,229.61,0.00),v40,z0,tPen\WObj:=wPaper;
    MoveL Offs(pOrigin,187.31,229.82,0.00),v40,z0,tPen\WObj:=wPaper;
    MoveL Offs(pOrigin,186.89,229.61,0.00),v40,z0,tPen\WObj:=wPaper;
    MoveL Offs(pOrigin,185.78,229.64,0.00),v40,z0,tPen\WObj:=wPaper;
    MoveL Offs(pOrigin,187.43,227.98,0.00),v40,z0,tPen\WObj:=wPaper;
    MoveL Offs(pOrigin,186.39,227.54,0.00),v40,z0,tPen\WObj:=wPaper;
    MoveL Offs(pOrigin,184.73,229.19,0.00),v40,z0,tPen\WObj:=wPaper;
    MoveL Offs(pOrigin,185.67,229.27,0.00),v40,z0,tPen\WObj:=wPaper;
    MoveL Offs(pOrigin,182.36,225.96,0.00),v40,z0,tPen\WObj:=wPaper;
    MoveL Offs(pOrigin,182.50,225.45,0.00),v40,z0,tPen\WObj:=wPaper;
    MoveL Offs(pOrigin,180.84,227.10,0.00),v40,z0,tPen\WObj:=wPaper;
    MoveL Offs(pOrigin,180.10,226.36,0.00),v40,z0,tPen\WObj:=wPaper;
    MoveL Offs(pOrigin,181.60,224.86,0.00),v40,z0,tPen\WObj:=wPaper;
    MoveL Offs(pOrigin,180.70,224.26,0.00),v40,z0,tPen\WObj:=wPaper;
    MoveL Offs(pOrigin,179.20,225.76,0.00),v40,z0,tPen\WObj:=wPaper;
    MoveL Offs(pOrigin,178.45,225.02,0.00),v40,z0,tPen\WObj:=wPaper;
    MoveL Offs(pOrigin,179.96,223.51,0.00),v40,z0,tPen\WObj:=wPaper;
    MoveL Offs(pOrigin,179.06,222.92,0.00),v40,z0,tPen\WObj:=wPaper;
    MoveL Offs(pOrigin,177.71,224.27,0.00),v40,z0,tPen\WObj:=wPaper;
    MoveL Offs(pOrigin,176.96,223.52,0.00),v40,z0,tPen\WObj:=wPaper;
    MoveL Offs(pOrigin,178.31,222.17,0.00),v40,z0,tPen\WObj:=wPaper;
    MoveL Offs(pOrigin,177.71,222.80,0.00),v40,z0,tPen\WObj:=wPaper;
    MoveL Offs(pOrigin,182.51,227.61,0.00),v40,z0,tPen\WObj:=wPaper;
    MoveL Offs(pOrigin,182.79,228.15,0.00),v40,z0,tPen\WObj:=wPaper;
    MoveL Offs(pOrigin,184.44,226.49,0.00),v40,z0,tPen\WObj:=wPaper;
    MoveL Offs(pOrigin,183.55,225.90,0.00),v40,z0,tPen\WObj:=wPaper;
    MoveL Offs(pOrigin,181.74,227.70,0.00),v40,fine,tPen\WObj:=wPaper;
    MoveL Offs(pOrigin,181.74,227.70,6.00),v60,z5,tPen\WObj:=wPaper;
    MoveL Offs(pOrigin,182.43,226.64,6.00),vTravel,z5,tPen\WObj:=wPaper;
    MoveL Offs(pOrigin,182.43,226.64,0.00),v60,z0,tPen\WObj:=wPaper;
    MoveL Offs(pOrigin,178.81,224.09,0.00),v40,z0,tPen\WObj:=wPaper;
    MoveL Offs(pOrigin,175.84,220.69,0.00),v40,z0,tPen\WObj:=wPaper;
    MoveL Offs(pOrigin,173.64,216.86,0.00),v40,z0,tPen\WObj:=wPaper;
    MoveL Offs(pOrigin,172.86,214.31,0.00),v40,z0,tPen\WObj:=wPaper;
    MoveL Offs(pOrigin,172.86,213.04,0.00),v40,fine,tPen\WObj:=wPaper;
    MoveL Offs(pOrigin,172.86,213.04,6.00),v60,z5,tPen\WObj:=wPaper;
    MoveL Offs(pOrigin,173.84,216.19,6.00),vTravel,z5,tPen\WObj:=wPaper;
    MoveL Offs(pOrigin,173.84,216.19,0.00),v60,z0,tPen\WObj:=wPaper;
    MoveL Offs(pOrigin,173.09,216.94,0.00),v40,z0,tPen\WObj:=wPaper;
    MoveL Offs(pOrigin,173.53,217.99,0.00),v40,z0,tPen\WObj:=wPaper;
    MoveL Offs(pOrigin,174.43,217.09,0.00),v40,z0,tPen\WObj:=wPaper;
    MoveL Offs(pOrigin,174.88,218.14,0.00),v40,z0,tPen\WObj:=wPaper;
    MoveL Offs(pOrigin,173.98,219.04,0.00),v40,z0,tPen\WObj:=wPaper;
    MoveL Offs(pOrigin,174.43,220.08,0.00),v40,z0,tPen\WObj:=wPaper;
    MoveL Offs(pOrigin,175.48,219.03,0.00),v40,z0,tPen\WObj:=wPaper;
    MoveL Offs(pOrigin,176.07,219.93,0.00),v40,z0,tPen\WObj:=wPaper;
    MoveL Offs(pOrigin,175.02,220.98,0.00),v40,z0,tPen\WObj:=wPaper;
    MoveL Offs(pOrigin,175.62,221.88,0.00),v40,z0,tPen\WObj:=wPaper;
    MoveL Offs(pOrigin,176.82,220.68,0.00),v40,z0,tPen\WObj:=wPaper;
    MoveL Offs(pOrigin,177.57,221.42,0.00),v40,z0,tPen\WObj:=wPaper;
    MoveL Offs(pOrigin,176.21,222.77,0.00),v40,fine,tPen\WObj:=wPaper;
    MoveL Offs(pOrigin,176.21,222.77,6.00),v60,z5,tPen\WObj:=wPaper;
    MoveL Offs(pOrigin,173.21,225.78,6.00),vTravel,z5,tPen\WObj:=wPaper;
    MoveL Offs(pOrigin,173.21,225.78,0.00),v60,z0,tPen\WObj:=wPaper;
    MoveL Offs(pOrigin,168.10,230.89,0.00),v40,z0,tPen\WObj:=wPaper;
    MoveL Offs(pOrigin,169.04,231.10,0.00),v40,z0,tPen\WObj:=wPaper;
    MoveL Offs(pOrigin,169.68,231.52,0.00),v40,z0,tPen\WObj:=wPaper;
    MoveL Offs(pOrigin,169.04,231.10,0.00),v40,z0,tPen\WObj:=wPaper;
    MoveL Offs(pOrigin,169.00,231.49,0.00),v40,z0,tPen\WObj:=wPaper;
    MoveL Offs(pOrigin,173.96,226.53,0.00),v40,z0,tPen\WObj:=wPaper;
    MoveL Offs(pOrigin,173.71,227.49,0.00),v40,z0,tPen\WObj:=wPaper;
    MoveL Offs(pOrigin,174.56,228.34,0.00),v40,z0,tPen\WObj:=wPaper;
    MoveL Offs(pOrigin,173.71,227.49,0.00),v40,z0,tPen\WObj:=wPaper;
    MoveL Offs(pOrigin,173.08,227.26,0.00),v40,z0,tPen\WObj:=wPaper;
    MoveL Offs(pOrigin,171.80,227.26,0.00),v40,z0,tPen\WObj:=wPaper;
    MoveL Offs(pOrigin,172.01,228.12,0.00),v40,z0,tPen\WObj:=wPaper;
    MoveL Offs(pOrigin,172.65,228.76,0.00),v40,z0,tPen\WObj:=wPaper;
    MoveL Offs(pOrigin,172.01,228.12,0.00),v40,z0,tPen\WObj:=wPaper;
    MoveL Offs(pOrigin,172.65,228.31,0.00),v40,z0,tPen\WObj:=wPaper;
    MoveL Offs(pOrigin,173.92,228.31,0.00),v40,z0,tPen\WObj:=wPaper;
  ENDPROC

  PROC DrawPart158()
    MoveL Offs(pOrigin,174.55,227.42,0.00),v40,z0,tPen\WObj:=wPaper;
    MoveL Offs(pOrigin,169.74,232.23,0.00),v40,z0,tPen\WObj:=wPaper;
    MoveL Offs(pOrigin,170.52,231.48,0.00),v40,z0,tPen\WObj:=wPaper;
    MoveL Offs(pOrigin,172.65,231.48,0.00),v40,z0,tPen\WObj:=wPaper;
    MoveL Offs(pOrigin,172.49,231.02,0.00),v40,z0,tPen\WObj:=wPaper;
    MoveL Offs(pOrigin,176.70,235.23,0.00),v40,z0,tPen\WObj:=wPaper;
    MoveL Offs(pOrigin,176.92,235.51,0.00),v40,z0,tPen\WObj:=wPaper;
    MoveL Offs(pOrigin,180.83,231.60,0.00),v40,z0,tPen\WObj:=wPaper;
    MoveL Offs(pOrigin,181.03,232.10,0.00),v40,z0,tPen\WObj:=wPaper;
    MoveL Offs(pOrigin,186.89,237.96,0.00),v40,z0,tPen\WObj:=wPaper;
    MoveL Offs(pOrigin,186.35,238.02,0.00),v40,z0,tPen\WObj:=wPaper;
    MoveL Offs(pOrigin,188.76,235.62,0.00),v40,z0,tPen\WObj:=wPaper;
    MoveL Offs(pOrigin,187.93,236.02,0.00),v40,z0,tPen\WObj:=wPaper;
    MoveL Offs(pOrigin,190.49,238.57,0.00),v40,z0,tPen\WObj:=wPaper;
    MoveL Offs(pOrigin,189.95,238.91,0.00),v40,z0,tPen\WObj:=wPaper;
    MoveL Offs(pOrigin,192.50,236.36,0.00),v40,fine,tPen\WObj:=wPaper;
    MoveL Offs(pOrigin,192.50,236.36,6.00),v60,z5,tPen\WObj:=wPaper;
    MoveL Offs(pOrigin,193.48,237.08,6.00),vTravel,z5,tPen\WObj:=wPaper;
    MoveL Offs(pOrigin,193.48,237.08,0.00),v60,z0,tPen\WObj:=wPaper;
    MoveL Offs(pOrigin,196.33,239.94,0.00),v40,z0,tPen\WObj:=wPaper;
    MoveL Offs(pOrigin,196.23,240.09,0.00),v40,z0,tPen\WObj:=wPaper;
    MoveL Offs(pOrigin,198.94,237.39,0.00),v40,z0,tPen\WObj:=wPaper;
    MoveL Offs(pOrigin,199.02,238.15,0.00),v40,z0,tPen\WObj:=wPaper;
    MoveL Offs(pOrigin,202.63,241.75,0.00),v40,z0,tPen\WObj:=wPaper;
    MoveL Offs(pOrigin,202.19,240.98,0.00),v40,z0,tPen\WObj:=wPaper;
    MoveL Offs(pOrigin,200.91,240.98,0.00),v40,z0,tPen\WObj:=wPaper;
    MoveL Offs(pOrigin,201.71,240.45,0.00),v40,z0,tPen\WObj:=wPaper;
    MoveL Offs(pOrigin,201.71,238.75,0.00),v40,z0,tPen\WObj:=wPaper;
    MoveL Offs(pOrigin,201.76,237.82,0.00),v40,z0,tPen\WObj:=wPaper;
    MoveL Offs(pOrigin,202.82,237.82,0.00),v40,z0,tPen\WObj:=wPaper;
    MoveL Offs(pOrigin,203.37,238.01,0.00),v40,z0,tPen\WObj:=wPaper;
    MoveL Offs(pOrigin,201.72,236.36,0.00),v40,fine,tPen\WObj:=wPaper;
    MoveL Offs(pOrigin,201.72,236.36,6.00),v60,z5,tPen\WObj:=wPaper;
    MoveL Offs(pOrigin,201.42,237.55,6.00),vTravel,z5,tPen\WObj:=wPaper;
    MoveL Offs(pOrigin,201.42,237.55,0.00),v60,z0,tPen\WObj:=wPaper;
    MoveL Offs(pOrigin,203.22,239.36,0.00),v40,z0,tPen\WObj:=wPaper;
    MoveL Offs(pOrigin,202.82,238.87,0.00),v40,z0,tPen\WObj:=wPaper;
    MoveL Offs(pOrigin,194.54,238.87,0.00),v40,z0,tPen\WObj:=wPaper;
    MoveL Offs(pOrigin,193.69,239.65,0.00),v40,z0,tPen\WObj:=wPaper;
    MoveL Offs(pOrigin,196.39,236.94,0.00),v40,z0,tPen\WObj:=wPaper;
    MoveL Offs(pOrigin,195.60,237.82,0.00),v40,z0,tPen\WObj:=wPaper;
    MoveL Offs(pOrigin,188.80,237.82,0.00),v40,fine,tPen\WObj:=wPaper;
    MoveL Offs(pOrigin,188.80,237.82,6.00),v60,z5,tPen\WObj:=wPaper;
    MoveL Offs(pOrigin,187.40,238.47,6.00),vTravel,z5,tPen\WObj:=wPaper;
    MoveL Offs(pOrigin,187.40,238.47,0.00),v60,z0,tPen\WObj:=wPaper;
    MoveL Offs(pOrigin,189.96,235.92,0.00),v40,fine,tPen\WObj:=wPaper;
    MoveL Offs(pOrigin,189.96,235.92,6.00),v60,z5,tPen\WObj:=wPaper;
    MoveL Offs(pOrigin,187.71,235.17,6.00),vTravel,z5,tPen\WObj:=wPaper;
    MoveL Offs(pOrigin,187.71,235.17,0.00),v60,z0,tPen\WObj:=wPaper;
    MoveL Offs(pOrigin,185.01,237.88,0.00),v40,z0,tPen\WObj:=wPaper;
    MoveL Offs(pOrigin,185.09,237.65,0.00),v40,z0,tPen\WObj:=wPaper;
    MoveL Offs(pOrigin,178.93,231.49,0.00),v40,z0,tPen\WObj:=wPaper;
    MoveL Offs(pOrigin,178.39,231.48,0.00),v40,z0,tPen\WObj:=wPaper;
    MoveL Offs(pOrigin,176.26,231.48,0.00),v40,fine,tPen\WObj:=wPaper;
    MoveL Offs(pOrigin,176.26,231.48,6.00),v60,z5,tPen\WObj:=wPaper;
    MoveL Offs(pOrigin,174.99,232.54,6.00),vTravel,z5,tPen\WObj:=wPaper;
    MoveL Offs(pOrigin,174.99,232.54,0.00),v60,z0,tPen\WObj:=wPaper;
    MoveL Offs(pOrigin,172.23,232.54,0.00),v40,z0,tPen\WObj:=wPaper;
    MoveL Offs(pOrigin,171.59,232.59,0.00),v40,z0,tPen\WObj:=wPaper;
    MoveL Offs(pOrigin,172.23,233.01,0.00),v40,z0,tPen\WObj:=wPaper;
    MoveL Offs(pOrigin,171.59,232.59,0.00),v40,z0,tPen\WObj:=wPaper;
    MoveL Offs(pOrigin,171.69,233.27,0.00),v40,z0,tPen\WObj:=wPaper;
    MoveL Offs(pOrigin,176.05,228.92,0.00),v40,fine,tPen\WObj:=wPaper;
    MoveL Offs(pOrigin,176.05,228.92,6.00),v60,z5,tPen\WObj:=wPaper;
    MoveL Offs(pOrigin,173.99,231.03,6.00),vTravel,z5,tPen\WObj:=wPaper;
    MoveL Offs(pOrigin,173.99,231.03,0.00),v60,z0,tPen\WObj:=wPaper;
    MoveL Offs(pOrigin,178.94,235.99,0.00),v40,z0,tPen\WObj:=wPaper;
    MoveL Offs(pOrigin,179.17,236.25,0.00),v40,z0,tPen\WObj:=wPaper;
    MoveL Offs(pOrigin,182.93,232.49,0.00),v40,z0,tPen\WObj:=wPaper;
    MoveL Offs(pOrigin,181.88,232.05,0.00),v40,z0,tPen\WObj:=wPaper;
    MoveL Offs(pOrigin,177.97,235.95,0.00),v40,fine,tPen\WObj:=wPaper;
    MoveL Offs(pOrigin,177.97,235.95,6.00),v60,z5,tPen\WObj:=wPaper;
    MoveL Offs(pOrigin,177.11,234.65,6.00),vTravel,z5,tPen\WObj:=wPaper;
    MoveL Offs(pOrigin,177.11,234.65,0.00),v60,z0,tPen\WObj:=wPaper;
    MoveL Offs(pOrigin,182.21,234.65,0.00),v40,fine,tPen\WObj:=wPaper;
    MoveL Offs(pOrigin,182.21,234.65,6.00),v60,z5,tPen\WObj:=wPaper;
    MoveL Offs(pOrigin,180.30,232.54,6.00),vTravel,z5,tPen\WObj:=wPaper;
    MoveL Offs(pOrigin,180.30,232.54,0.00),v60,z0,tPen\WObj:=wPaper;
    MoveL Offs(pOrigin,178.18,232.54,0.00),v40,z0,tPen\WObj:=wPaper;
    MoveL Offs(pOrigin,177.96,232.59,0.00),v40,z0,tPen\WObj:=wPaper;
    MoveL Offs(pOrigin,178.39,232.80,0.00),v40,z0,tPen\WObj:=wPaper;
    MoveL Offs(pOrigin,177.96,232.59,0.00),v40,fine,tPen\WObj:=wPaper;
    MoveL Offs(pOrigin,177.96,232.59,6.00),v60,z5,tPen\WObj:=wPaper;
    MoveL Offs(pOrigin,178.81,233.59,6.00),vTravel,z5,tPen\WObj:=wPaper;
    MoveL Offs(pOrigin,178.81,233.59,0.00),v60,z0,tPen\WObj:=wPaper;
    MoveL Offs(pOrigin,174.56,233.59,0.00),v40,fine,tPen\WObj:=wPaper;
    MoveL Offs(pOrigin,174.56,233.59,6.00),v60,z5,tPen\WObj:=wPaper;
    MoveL Offs(pOrigin,175.88,235.06,6.00),vTravel,z5,tPen\WObj:=wPaper;
    MoveL Offs(pOrigin,175.88,235.06,0.00),v60,z0,tPen\WObj:=wPaper;
    MoveL Offs(pOrigin,179.63,231.30,0.00),v40,fine,tPen\WObj:=wPaper;
    MoveL Offs(pOrigin,179.63,231.30,6.00),v60,z5,tPen\WObj:=wPaper;
    MoveL Offs(pOrigin,183.69,228.74,6.00),vTravel,z5,tPen\WObj:=wPaper;
    MoveL Offs(pOrigin,183.69,228.74,0.00),v60,z0,tPen\WObj:=wPaper;
    MoveL Offs(pOrigin,185.49,226.94,0.00),v40,z0,tPen\WObj:=wPaper;
    MoveL Offs(pOrigin,185.66,227.77,0.00),v40,z0,tPen\WObj:=wPaper;
    MoveL Offs(pOrigin,188.37,230.47,0.00),v40,z0,tPen\WObj:=wPaper;
    MoveL Offs(pOrigin,187.72,230.68,0.00),v40,z0,tPen\WObj:=wPaper;
    MoveL Offs(pOrigin,189.68,228.73,0.00),v40,z0,tPen\WObj:=wPaper;
    MoveL Offs(pOrigin,190.46,229.58,0.00),v40,z0,tPen\WObj:=wPaper;
    MoveL Offs(pOrigin,193.16,232.29,0.00),v40,z0,tPen\WObj:=wPaper;
    MoveL Offs(pOrigin,193.41,232.46,0.00),v40,z0,tPen\WObj:=wPaper;
    MoveL Offs(pOrigin,195.37,230.51,0.00),v40,z0,tPen\WObj:=wPaper;
    MoveL Offs(pOrigin,194.81,230.94,0.00),v40,z0,tPen\WObj:=wPaper;
    MoveL Offs(pOrigin,197.21,233.35,0.00),v40,z0,tPen\WObj:=wPaper;
    MoveL Offs(pOrigin,196.70,233.65,0.00),v40,z0,tPen\WObj:=wPaper;
    MoveL Offs(pOrigin,198.96,231.39,0.00),v40,z0,tPen\WObj:=wPaper;
    MoveL Offs(pOrigin,198.86,232.00,0.00),v40,z0,tPen\WObj:=wPaper;
    MoveL Offs(pOrigin,203.66,236.81,0.00),v40,z0,tPen\WObj:=wPaper;
    MoveL Offs(pOrigin,204.03,236.77,0.00),v40,z0,tPen\WObj:=wPaper;
    MoveL Offs(pOrigin,199.68,241.13,0.00),v40,z0,tPen\WObj:=wPaper;
    MoveL Offs(pOrigin,198.78,240.53,0.00),v40,z0,tPen\WObj:=wPaper;
    MoveL Offs(pOrigin,204.19,235.12,0.00),v40,z0,tPen\WObj:=wPaper;
    MoveL Offs(pOrigin,203.81,235.46,0.00),v40,z0,tPen\WObj:=wPaper;
    MoveL Offs(pOrigin,200.50,232.16,0.00),v40,z0,tPen\WObj:=wPaper;
    MoveL Offs(pOrigin,200.31,231.54,0.00),v40,z0,tPen\WObj:=wPaper;
    MoveL Offs(pOrigin,198.05,233.79,0.00),v40,fine,tPen\WObj:=wPaper;
    MoveL Offs(pOrigin,198.05,233.79,6.00),v60,z5,tPen\WObj:=wPaper;
    MoveL Offs(pOrigin,200.45,234.38,6.00),vTravel,z5,tPen\WObj:=wPaper;
    MoveL Offs(pOrigin,200.45,234.38,0.00),v60,z0,tPen\WObj:=wPaper;
    MoveL Offs(pOrigin,212.47,222.36,0.00),v40,fine,tPen\WObj:=wPaper;
  ENDPROC

  PROC DrawPart159()
    MoveL Offs(pOrigin,212.47,222.36,6.00),v60,z5,tPen\WObj:=wPaper;
    MoveL Offs(pOrigin,212.90,220.66,6.00),vTravel,z5,tPen\WObj:=wPaper;
    MoveL Offs(pOrigin,212.90,220.66,0.00),v60,z0,tPen\WObj:=wPaper;
    MoveL Offs(pOrigin,211.40,219.16,0.00),v40,fine,tPen\WObj:=wPaper;
    MoveL Offs(pOrigin,211.40,219.16,6.00),v60,z5,tPen\WObj:=wPaper;
    MoveL Offs(pOrigin,212.81,220.05,6.00),vTravel,z5,tPen\WObj:=wPaper;
    MoveL Offs(pOrigin,212.81,220.05,0.00),v60,z0,tPen\WObj:=wPaper;
    MoveL Offs(pOrigin,212.39,220.69,0.00),v40,z0,tPen\WObj:=wPaper;
    MoveL Offs(pOrigin,212.81,220.05,0.00),v40,fine,tPen\WObj:=wPaper;
    MoveL Offs(pOrigin,212.81,220.05,6.00),v60,z5,tPen\WObj:=wPaper;
    MoveL Offs(pOrigin,209.93,220.42,6.00),vTravel,z5,tPen\WObj:=wPaper;
    MoveL Offs(pOrigin,209.93,220.42,0.00),v60,z0,tPen\WObj:=wPaper;
    MoveL Offs(pOrigin,232.47,197.89,0.00),v40,z0,tPen\WObj:=wPaper;
    MoveL Offs(pOrigin,231.86,197.80,0.00),v40,z0,tPen\WObj:=wPaper;
    MoveL Offs(pOrigin,229.90,195.85,0.00),v40,z0,tPen\WObj:=wPaper;
    MoveL Offs(pOrigin,230.02,196.63,0.00),v40,z0,tPen\WObj:=wPaper;
    MoveL Offs(pOrigin,232.36,196.63,0.00),v40,z0,tPen\WObj:=wPaper;
    MoveL Offs(pOrigin,232.60,197.05,0.00),v40,z0,tPen\WObj:=wPaper;
    MoveL Offs(pOrigin,230.50,194.95,0.00),v40,z0,tPen\WObj:=wPaper;
    MoveL Offs(pOrigin,230.88,194.98,0.00),v40,z0,tPen\WObj:=wPaper;
    MoveL Offs(pOrigin,230.66,195.40,0.00),v40,z0,tPen\WObj:=wPaper;
    MoveL Offs(pOrigin,230.88,194.98,0.00),v40,z0,tPen\WObj:=wPaper;
    MoveL Offs(pOrigin,231.28,195.19,0.00),v40,z0,tPen\WObj:=wPaper;
    MoveL Offs(pOrigin,231.28,197.10,0.00),v40,z0,tPen\WObj:=wPaper;
    MoveL Offs(pOrigin,231.73,197.10,0.00),v40,z0,tPen\WObj:=wPaper;
    MoveL Offs(pOrigin,231.30,197.52,0.00),v40,z0,tPen\WObj:=wPaper;
    MoveL Offs(pOrigin,231.73,197.10,0.00),v40,z0,tPen\WObj:=wPaper;
    MoveL Offs(pOrigin,231.30,197.69,0.00),v40,z0,tPen\WObj:=wPaper;
    MoveL Offs(pOrigin,229.39,197.69,0.00),v40,z0,tPen\WObj:=wPaper;
    MoveL Offs(pOrigin,229.39,197.52,0.00),v40,z0,tPen\WObj:=wPaper;
    MoveL Offs(pOrigin,228.96,198.16,0.00),v40,z0,tPen\WObj:=wPaper;
    MoveL Offs(pOrigin,229.39,197.52,0.00),v40,z0,tPen\WObj:=wPaper;
    MoveL Offs(pOrigin,228.86,197.79,0.00),v40,z0,tPen\WObj:=wPaper;
    MoveL Offs(pOrigin,230.36,199.29,0.00),v40,z0,tPen\WObj:=wPaper;
    MoveL Offs(pOrigin,230.45,198.74,0.00),v40,z0,tPen\WObj:=wPaper;
    MoveL Offs(pOrigin,228.75,198.74,0.00),v40,z0,tPen\WObj:=wPaper;
    MoveL Offs(pOrigin,228.75,198.59,0.00),v40,z0,tPen\WObj:=wPaper;
    MoveL Offs(pOrigin,228.32,199.23,0.00),v40,z0,tPen\WObj:=wPaper;
    MoveL Offs(pOrigin,228.75,198.59,0.00),v40,z0,tPen\WObj:=wPaper;
    MoveL Offs(pOrigin,228.26,198.69,0.00),v40,z0,tPen\WObj:=wPaper;
    MoveL Offs(pOrigin,231.72,202.15,0.00),v40,z0,tPen\WObj:=wPaper;
    MoveL Offs(pOrigin,232.47,201.40,0.00),v40,z0,tPen\WObj:=wPaper;
    MoveL Offs(pOrigin,231.42,200.35,0.00),v40,z0,tPen\WObj:=wPaper;
    MoveL Offs(pOrigin,232.46,199.90,0.00),v40,z0,tPen\WObj:=wPaper;
    MoveL Offs(pOrigin,233.36,200.80,0.00),v40,z0,tPen\WObj:=wPaper;
    MoveL Offs(pOrigin,233.35,201.48,0.00),v40,z0,tPen\WObj:=wPaper;
    MoveL Offs(pOrigin,237.71,197.12,0.00),v40,fine,tPen\WObj:=wPaper;
    MoveL Offs(pOrigin,237.71,197.12,6.00),v60,z5,tPen\WObj:=wPaper;
    MoveL Offs(pOrigin,239.36,196.97,6.00),vTravel,z5,tPen\WObj:=wPaper;
    MoveL Offs(pOrigin,239.36,196.97,0.00),v60,z0,tPen\WObj:=wPaper;
    MoveL Offs(pOrigin,236.80,199.52,0.00),v40,fine,tPen\WObj:=wPaper;
    MoveL Offs(pOrigin,236.80,199.52,6.00),v60,z5,tPen\WObj:=wPaper;
    MoveL Offs(pOrigin,235.46,197.88,6.00),vTravel,z5,tPen\WObj:=wPaper;
    MoveL Offs(pOrigin,235.46,197.88,0.00),v60,z0,tPen\WObj:=wPaper;
    MoveL Offs(pOrigin,228.25,205.09,0.00),v40,z0,tPen\WObj:=wPaper;
    MoveL Offs(pOrigin,228.28,204.68,0.00),v40,z0,tPen\WObj:=wPaper;
    MoveL Offs(pOrigin,226.03,202.43,0.00),v40,z0,tPen\WObj:=wPaper;
    MoveL Offs(pOrigin,226.41,202.41,0.00),v40,z0,tPen\WObj:=wPaper;
    MoveL Offs(pOrigin,226.20,202.84,0.00),v40,z0,tPen\WObj:=wPaper;
    MoveL Offs(pOrigin,226.41,202.41,0.00),v40,z0,tPen\WObj:=wPaper;
    MoveL Offs(pOrigin,226.20,202.97,0.00),v40,z0,tPen\WObj:=wPaper;
    MoveL Offs(pOrigin,229.18,202.97,0.00),v40,z0,tPen\WObj:=wPaper;
    MoveL Offs(pOrigin,229.39,202.62,0.00),v40,z0,tPen\WObj:=wPaper;
    MoveL Offs(pOrigin,229.10,203.40,0.00),v40,z0,tPen\WObj:=wPaper;
    MoveL Offs(pOrigin,228.54,203.55,0.00),v40,z0,tPen\WObj:=wPaper;
    MoveL Offs(pOrigin,228.11,202.84,0.00),v40,z0,tPen\WObj:=wPaper;
    MoveL Offs(pOrigin,228.32,202.41,0.00),v40,z0,tPen\WObj:=wPaper;
    MoveL Offs(pOrigin,228.11,203.26,0.00),v40,z0,tPen\WObj:=wPaper;
    MoveL Offs(pOrigin,228.32,203.69,0.00),v40,z0,tPen\WObj:=wPaper;
    MoveL Offs(pOrigin,228.11,203.26,0.00),v40,z0,tPen\WObj:=wPaper;
    MoveL Offs(pOrigin,228.32,203.69,0.00),v40,z0,tPen\WObj:=wPaper;
    MoveL Offs(pOrigin,222.38,209.64,0.00),v40,z0,tPen\WObj:=wPaper;
    MoveL Offs(pOrigin,221.95,210.91,0.00),v40,z0,tPen\WObj:=wPaper;
    MoveL Offs(pOrigin,222.16,210.36,0.00),v40,z0,tPen\WObj:=wPaper;
    MoveL Offs(pOrigin,219.40,210.36,0.00),v40,z0,tPen\WObj:=wPaper;
    MoveL Offs(pOrigin,219.01,210.35,0.00),v40,z0,tPen\WObj:=wPaper;
    MoveL Offs(pOrigin,221.27,212.60,0.00),v40,z0,tPen\WObj:=wPaper;
    MoveL Offs(pOrigin,220.46,212.47,0.00),v40,z0,tPen\WObj:=wPaper;
    MoveL Offs(pOrigin,208.14,212.47,0.00),v40,z0,tPen\WObj:=wPaper;
    MoveL Offs(pOrigin,208.00,213.39,0.00),v40,z0,tPen\WObj:=wPaper;
    MoveL Offs(pOrigin,210.71,210.69,0.00),v40,z0,tPen\WObj:=wPaper;
    MoveL Offs(pOrigin,211.08,211.37,0.00),v40,z0,tPen\WObj:=wPaper;
    MoveL Offs(pOrigin,213.63,213.92,0.00),v40,z0,tPen\WObj:=wPaper;
    MoveL Offs(pOrigin,213.09,214.27,0.00),v40,z0,tPen\WObj:=wPaper;
    MoveL Offs(pOrigin,217.00,210.37,0.00),v40,z0,tPen\WObj:=wPaper;
    MoveL Offs(pOrigin,216.43,210.91,0.00),v40,z0,tPen\WObj:=wPaper;
    MoveL Offs(pOrigin,217.27,211.76,0.00),v40,z0,tPen\WObj:=wPaper;
    MoveL Offs(pOrigin,216.43,210.91,0.00),v40,z0,tPen\WObj:=wPaper;
    MoveL Offs(pOrigin,217.06,211.42,0.00),v40,z0,tPen\WObj:=wPaper;
    MoveL Offs(pOrigin,214.51,211.42,0.00),v40,z0,tPen\WObj:=wPaper;
    MoveL Offs(pOrigin,215.44,211.12,0.00),v40,z0,tPen\WObj:=wPaper;
    MoveL Offs(pOrigin,215.44,213.46,0.00),v40,z0,tPen\WObj:=wPaper;
    MoveL Offs(pOrigin,214.72,213.53,0.00),v40,z0,tPen\WObj:=wPaper;
    MoveL Offs(pOrigin,218.98,213.53,0.00),v40,z0,tPen\WObj:=wPaper;
    MoveL Offs(pOrigin,219.47,213.79,0.00),v40,z0,tPen\WObj:=wPaper;
    MoveL Offs(pOrigin,196.33,190.65,0.00),v40,z0,tPen\WObj:=wPaper;
    MoveL Offs(pOrigin,196.88,190.73,0.00),v40,z0,tPen\WObj:=wPaper;
    MoveL Offs(pOrigin,197.51,191.36,0.00),v40,z0,tPen\WObj:=wPaper;
    MoveL Offs(pOrigin,196.88,190.73,0.00),v40,z0,tPen\WObj:=wPaper;
    MoveL Offs(pOrigin,196.88,190.30,0.00),v40,z0,tPen\WObj:=wPaper;
    MoveL Offs(pOrigin,198.58,190.30,0.00),v40,z0,tPen\WObj:=wPaper;
    MoveL Offs(pOrigin,199.48,190.81,0.00),v40,z0,tPen\WObj:=wPaper;
    MoveL Offs(pOrigin,197.07,188.41,0.00),v40,z0,tPen\WObj:=wPaper;
    MoveL Offs(pOrigin,196.88,189.24,0.00),v40,z0,tPen\WObj:=wPaper;
    MoveL Offs(pOrigin,199.00,189.24,0.00),v40,z0,tPen\WObj:=wPaper;
    MoveL Offs(pOrigin,199.62,189.46,0.00),v40,z0,tPen\WObj:=wPaper;
    MoveL Offs(pOrigin,198.12,187.96,0.00),v40,z0,tPen\WObj:=wPaper;
    MoveL Offs(pOrigin,198.36,188.18,0.00),v40,z0,tPen\WObj:=wPaper;
    MoveL Offs(pOrigin,201.34,188.18,0.00),v40,z0,tPen\WObj:=wPaper;
    MoveL Offs(pOrigin,201.87,188.72,0.00),v40,z0,tPen\WObj:=wPaper;
    MoveL Offs(pOrigin,200.37,187.22,0.00),v40,z0,tPen\WObj:=wPaper;
    MoveL Offs(pOrigin,201.34,187.13,0.00),v40,z0,tPen\WObj:=wPaper;
    MoveL Offs(pOrigin,204.52,187.13,0.00),v40,z0,tPen\WObj:=wPaper;
    MoveL Offs(pOrigin,204.11,187.98,0.00),v40,z0,tPen\WObj:=wPaper;
    MoveL Offs(pOrigin,202.61,186.48,0.00),v40,z0,tPen\WObj:=wPaper;
    MoveL Offs(pOrigin,203.66,186.03,0.00),v40,z0,tPen\WObj:=wPaper;
    MoveL Offs(pOrigin,205.31,187.68,0.00),v40,z0,tPen\WObj:=wPaper;
    MoveL Offs(pOrigin,204.93,188.08,0.00),v40,z0,tPen\WObj:=wPaper;
    MoveL Offs(pOrigin,209.29,183.73,0.00),v40,z0,tPen\WObj:=wPaper;
    MoveL Offs(pOrigin,208.99,184.77,0.00),v40,z0,tPen\WObj:=wPaper;
  ENDPROC

  PROC DrawPart160()
    MoveL Offs(pOrigin,209.41,184.99,0.00),v40,z0,tPen\WObj:=wPaper;
    MoveL Offs(pOrigin,208.99,184.77,0.00),v40,z0,tPen\WObj:=wPaper;
    MoveL Offs(pOrigin,209.62,185.02,0.00),v40,z0,tPen\WObj:=wPaper;
    MoveL Offs(pOrigin,206.01,185.02,0.00),v40,z0,tPen\WObj:=wPaper;
    MoveL Offs(pOrigin,206.99,184.56,0.00),v40,z0,tPen\WObj:=wPaper;
    MoveL Offs(pOrigin,206.99,185.84,0.00),v40,z0,tPen\WObj:=wPaper;
    MoveL Offs(pOrigin,207.92,186.07,0.00),v40,z0,tPen\WObj:=wPaper;
    MoveL Offs(pOrigin,204.31,186.07,0.00),v40,z0,tPen\WObj:=wPaper;
    MoveL Offs(pOrigin,204.71,185.58,0.00),v40,z0,tPen\WObj:=wPaper;
    MoveL Offs(pOrigin,206.36,187.24,0.00),v40,fine,tPen\WObj:=wPaper;
    MoveL Offs(pOrigin,206.36,187.24,6.00),v60,z5,tPen\WObj:=wPaper;
    MoveL Offs(pOrigin,208.75,186.65,6.00),vTravel,z5,tPen\WObj:=wPaper;
    MoveL Offs(pOrigin,208.75,186.65,0.00),v60,z0,tPen\WObj:=wPaper;
    MoveL Offs(pOrigin,203.04,180.94,0.00),v40,z0,tPen\WObj:=wPaper;
    MoveL Offs(pOrigin,202.82,181.38,0.00),v40,z0,tPen\WObj:=wPaper;
    MoveL Offs(pOrigin,203.25,181.59,0.00),v40,z0,tPen\WObj:=wPaper;
    MoveL Offs(pOrigin,202.82,181.38,0.00),v40,z0,tPen\WObj:=wPaper;
    MoveL Offs(pOrigin,201.98,180.95,0.00),v40,z0,tPen\WObj:=wPaper;
    MoveL Offs(pOrigin,202.40,181.16,0.00),v40,z0,tPen\WObj:=wPaper;
    MoveL Offs(pOrigin,201.98,180.95,0.00),v40,z0,tPen\WObj:=wPaper;
    MoveL Offs(pOrigin,201.98,180.79,0.00),v40,z0,tPen\WObj:=wPaper;
    MoveL Offs(pOrigin,199.85,180.79,0.00),v40,z0,tPen\WObj:=wPaper;
    MoveL Offs(pOrigin,199.64,181.16,0.00),v40,z0,tPen\WObj:=wPaper;
    MoveL Offs(pOrigin,200.06,181.38,0.00),v40,z0,tPen\WObj:=wPaper;
    MoveL Offs(pOrigin,199.64,181.16,0.00),v40,z0,tPen\WObj:=wPaper;
    MoveL Offs(pOrigin,199.41,181.66,0.00),v40,z0,tPen\WObj:=wPaper;
    MoveL Offs(pOrigin,201.51,179.56,0.00),v40,z0,tPen\WObj:=wPaper;
    MoveL Offs(pOrigin,200.91,180.31,0.00),v40,z0,tPen\WObj:=wPaper;
    MoveL Offs(pOrigin,201.34,180.52,0.00),v40,z0,tPen\WObj:=wPaper;
    MoveL Offs(pOrigin,200.91,180.31,0.00),v40,fine,tPen\WObj:=wPaper;
    MoveL Offs(pOrigin,200.91,180.31,6.00),v60,z5,tPen\WObj:=wPaper;
    MoveL Offs(pOrigin,199.85,179.74,6.00),vTravel,z5,tPen\WObj:=wPaper;
    MoveL Offs(pOrigin,199.85,179.74,0.00),v60,z0,tPen\WObj:=wPaper;
    MoveL Offs(pOrigin,197.73,179.74,0.00),v40,z0,tPen\WObj:=wPaper;
    MoveL Offs(pOrigin,197.30,179.89,0.00),v40,z0,tPen\WObj:=wPaper;
    MoveL Offs(pOrigin,197.73,180.10,0.00),v40,z0,tPen\WObj:=wPaper;
    MoveL Offs(pOrigin,197.30,179.89,0.00),v40,z0,tPen\WObj:=wPaper;
    MoveL Offs(pOrigin,197.32,180.77,0.00),v40,z0,tPen\WObj:=wPaper;
    MoveL Offs(pOrigin,199.57,178.51,0.00),v40,z0,tPen\WObj:=wPaper;
    MoveL Offs(pOrigin,198.79,179.25,0.00),v40,z0,tPen\WObj:=wPaper;
    MoveL Offs(pOrigin,199.21,179.46,0.00),v40,z0,tPen\WObj:=wPaper;
    MoveL Offs(pOrigin,198.79,179.25,0.00),v40,z0,tPen\WObj:=wPaper;
    MoveL Offs(pOrigin,199.64,179.68,0.00),v40,z0,tPen\WObj:=wPaper;
    MoveL Offs(pOrigin,200.06,179.89,0.00),v40,z0,tPen\WObj:=wPaper;
    MoveL Offs(pOrigin,199.64,179.68,0.00),v40,fine,tPen\WObj:=wPaper;
    MoveL Offs(pOrigin,199.64,179.68,6.00),v60,z5,tPen\WObj:=wPaper;
    MoveL Offs(pOrigin,198.15,180.31,6.00),vTravel,z5,tPen\WObj:=wPaper;
    MoveL Offs(pOrigin,198.15,180.31,0.00),v60,z0,tPen\WObj:=wPaper;
    MoveL Offs(pOrigin,198.79,180.74,0.00),v40,z0,tPen\WObj:=wPaper;
    MoveL Offs(pOrigin,198.15,180.31,0.00),v40,fine,tPen\WObj:=wPaper;
    MoveL Offs(pOrigin,198.15,180.31,6.00),v60,z5,tPen\WObj:=wPaper;
    MoveL Offs(pOrigin,197.94,178.82,6.00),vTravel,z5,tPen\WObj:=wPaper;
    MoveL Offs(pOrigin,197.94,178.82,0.00),v60,z0,tPen\WObj:=wPaper;
    MoveL Offs(pOrigin,198.36,179.04,0.00),v40,z0,tPen\WObj:=wPaper;
    MoveL Offs(pOrigin,197.94,178.82,0.00),v40,z0,tPen\WObj:=wPaper;
    MoveL Offs(pOrigin,197.94,178.68,0.00),v40,z0,tPen\WObj:=wPaper;
    MoveL Offs(pOrigin,195.81,178.68,0.00),v40,z0,tPen\WObj:=wPaper;
    MoveL Offs(pOrigin,196.02,179.25,0.00),v40,z0,tPen\WObj:=wPaper;
    MoveL Offs(pOrigin,196.45,179.46,0.00),v40,z0,tPen\WObj:=wPaper;
    MoveL Offs(pOrigin,196.02,179.25,0.00),v40,z0,tPen\WObj:=wPaper;
    MoveL Offs(pOrigin,195.70,179.56,0.00),v40,z0,tPen\WObj:=wPaper;
    MoveL Offs(pOrigin,193.60,177.46,0.00),v40,z0,tPen\WObj:=wPaper;
    MoveL Offs(pOrigin,193.13,177.48,0.00),v40,z0,tPen\WObj:=wPaper;
    MoveL Offs(pOrigin,196.89,173.73,0.00),v40,z0,tPen\WObj:=wPaper;
    MoveL Offs(pOrigin,196.13,174.02,0.00),v40,z0,tPen\WObj:=wPaper;
    MoveL Offs(pOrigin,194.63,172.52,0.00),v40,z0,tPen\WObj:=wPaper;
    MoveL Offs(pOrigin,194.05,172.09,0.00),v40,z0,tPen\WObj:=wPaper;
    MoveL Offs(pOrigin,198.55,167.58,0.00),v40,z0,tPen\WObj:=wPaper;
    MoveL Offs(pOrigin,198.06,166.99,0.00),v40,z0,tPen\WObj:=wPaper;
    MoveL Offs(pOrigin,196.25,165.19,0.00),v40,z0,tPen\WObj:=wPaper;
    MoveL Offs(pOrigin,197.09,164.95,0.00),v40,z0,tPen\WObj:=wPaper;
    MoveL Offs(pOrigin,198.15,164.95,0.00),v40,z0,tPen\WObj:=wPaper;
    MoveL Offs(pOrigin,198.65,164.59,0.00),v40,z0,tPen\WObj:=wPaper;
    MoveL Offs(pOrigin,197.00,162.94,0.00),v40,z0,tPen\WObj:=wPaper;
    MoveL Offs(pOrigin,197.51,162.84,0.00),v40,z0,tPen\WObj:=wPaper;
    MoveL Offs(pOrigin,198.58,162.84,0.00),v40,z0,tPen\WObj:=wPaper;
    MoveL Offs(pOrigin,198.36,163.90,0.00),v40,z0,tPen\WObj:=wPaper;
    MoveL Offs(pOrigin,197.30,163.90,0.00),v40,fine,tPen\WObj:=wPaper;
    MoveL Offs(pOrigin,197.30,163.90,6.00),v60,z5,tPen\WObj:=wPaper;
    MoveL Offs(pOrigin,196.62,162.04,6.00),vTravel,z5,tPen\WObj:=wPaper;
    MoveL Offs(pOrigin,196.62,162.04,0.00),v60,z0,tPen\WObj:=wPaper;
    MoveL Offs(pOrigin,201.13,157.54,0.00),v40,z0,tPen\WObj:=wPaper;
    MoveL Offs(pOrigin,200.58,157.56,0.00),v40,z0,tPen\WObj:=wPaper;
    MoveL Offs(pOrigin,198.77,155.76,0.00),v40,z0,tPen\WObj:=wPaper;
    MoveL Offs(pOrigin,198.29,155.90,0.00),v40,z0,tPen\WObj:=wPaper;
    MoveL Offs(pOrigin,202.80,151.39,0.00),v40,fine,tPen\WObj:=wPaper;
    MoveL Offs(pOrigin,202.80,151.39,6.00),v60,z5,tPen\WObj:=wPaper;
    MoveL Offs(pOrigin,201.34,152.28,6.00),vTravel,z5,tPen\WObj:=wPaper;
    MoveL Offs(pOrigin,201.34,152.28,0.00),v60,z0,tPen\WObj:=wPaper;
    MoveL Offs(pOrigin,200.28,152.28,0.00),v40,z0,tPen\WObj:=wPaper;
    MoveL Offs(pOrigin,199.81,152.31,0.00),v40,z0,tPen\WObj:=wPaper;
    MoveL Offs(pOrigin,201.61,154.12,0.00),v40,z0,tPen\WObj:=wPaper;
    MoveL Offs(pOrigin,200.91,154.39,0.00),v40,z0,tPen\WObj:=wPaper;
    MoveL Offs(pOrigin,199.85,154.39,0.00),v40,z0,tPen\WObj:=wPaper;
    MoveL Offs(pOrigin,199.51,153.51,0.00),v40,z0,tPen\WObj:=wPaper;
    MoveL Offs(pOrigin,201.17,155.16,0.00),v40,z0,tPen\WObj:=wPaper;
    MoveL Offs(pOrigin,200.70,155.45,0.00),v40,z0,tPen\WObj:=wPaper;
    MoveL Offs(pOrigin,199.64,155.45,0.00),v40,fine,tPen\WObj:=wPaper;
    MoveL Offs(pOrigin,199.64,155.45,6.00),v60,z5,tPen\WObj:=wPaper;
    MoveL Offs(pOrigin,201.74,155.44,6.00),vTravel,z5,tPen\WObj:=wPaper;
    MoveL Offs(pOrigin,201.74,155.44,0.00),v60,z0,tPen\WObj:=wPaper;
    MoveL Offs(pOrigin,197.23,159.94,0.00),v40,fine,tPen\WObj:=wPaper;
    MoveL Offs(pOrigin,197.23,159.94,6.00),v60,z5,tPen\WObj:=wPaper;
    MoveL Offs(pOrigin,199.00,157.56,6.00),vTravel,z5,tPen\WObj:=wPaper;
    MoveL Offs(pOrigin,199.00,157.56,0.00),v60,z0,tPen\WObj:=wPaper;
    MoveL Offs(pOrigin,200.06,157.56,0.00),v40,fine,tPen\WObj:=wPaper;
    MoveL Offs(pOrigin,200.06,157.56,6.00),v60,z5,tPen\WObj:=wPaper;
    MoveL Offs(pOrigin,200.07,161.58,6.00),vTravel,z5,tPen\WObj:=wPaper;
    MoveL Offs(pOrigin,200.07,161.58,0.00),v60,z0,tPen\WObj:=wPaper;
    MoveL Offs(pOrigin,195.71,165.94,0.00),v40,z0,tPen\WObj:=wPaper;
    MoveL Offs(pOrigin,196.11,166.53,0.00),v40,z0,tPen\WObj:=wPaper;
    MoveL Offs(pOrigin,197.76,168.19,0.00),v40,z0,tPen\WObj:=wPaper;
    MoveL Offs(pOrigin,197.30,168.12,0.00),v40,z0,tPen\WObj:=wPaper;
    MoveL Offs(pOrigin,196.24,168.12,0.00),v40,z0,tPen\WObj:=wPaper;
    MoveL Offs(pOrigin,196.45,167.06,0.00),v40,z0,tPen\WObj:=wPaper;
    MoveL Offs(pOrigin,197.51,167.06,0.00),v40,fine,tPen\WObj:=wPaper;
    MoveL Offs(pOrigin,197.51,167.06,6.00),v60,z5,tPen\WObj:=wPaper;
    MoveL Offs(pOrigin,195.52,168.93,6.00),vTravel,z5,tPen\WObj:=wPaper;
    MoveL Offs(pOrigin,195.52,168.93,0.00),v60,z0,tPen\WObj:=wPaper;
    MoveL Offs(pOrigin,197.02,170.43,0.00),v40,z0,tPen\WObj:=wPaper;
  ENDPROC

  PROC DrawPart161()
    MoveL Offs(pOrigin,196.45,171.29,0.00),v40,z0,tPen\WObj:=wPaper;
    MoveL Offs(pOrigin,195.39,171.29,0.00),v40,z0,tPen\WObj:=wPaper;
    MoveL Offs(pOrigin,194.92,171.32,0.00),v40,z0,tPen\WObj:=wPaper;
    MoveL Offs(pOrigin,196.58,172.98,0.00),v40,fine,tPen\WObj:=wPaper;
    MoveL Offs(pOrigin,196.58,172.98,6.00),v60,z5,tPen\WObj:=wPaper;
    MoveL Offs(pOrigin,195.60,174.46,6.00),vTravel,z5,tPen\WObj:=wPaper;
    MoveL Offs(pOrigin,195.60,174.46,0.00),v60,z0,tPen\WObj:=wPaper;
    MoveL Offs(pOrigin,194.54,174.46,0.00),v40,z0,tPen\WObj:=wPaper;
    MoveL Offs(pOrigin,193.89,174.77,0.00),v40,z0,tPen\WObj:=wPaper;
    MoveL Offs(pOrigin,195.84,176.72,0.00),v40,z0,tPen\WObj:=wPaper;
    MoveL Offs(pOrigin,195.39,176.57,0.00),v40,z0,tPen\WObj:=wPaper;
    MoveL Offs(pOrigin,194.11,176.57,0.00),v40,z0,tPen\WObj:=wPaper;
    MoveL Offs(pOrigin,194.32,175.51,0.00),v40,z0,tPen\WObj:=wPaper;
    MoveL Offs(pOrigin,195.39,175.51,0.00),v40,fine,tPen\WObj:=wPaper;
    MoveL Offs(pOrigin,195.39,175.51,6.00),v60,z5,tPen\WObj:=wPaper;
    MoveL Offs(pOrigin,195.18,177.34,6.00),vTravel,z5,tPen\WObj:=wPaper;
    MoveL Offs(pOrigin,195.18,177.34,0.00),v60,z0,tPen\WObj:=wPaper;
    MoveL Offs(pOrigin,195.60,177.55,0.00),v40,z0,tPen\WObj:=wPaper;
    MoveL Offs(pOrigin,195.18,177.34,0.00),v40,fine,tPen\WObj:=wPaper;
    MoveL Offs(pOrigin,195.18,177.34,6.00),v60,z5,tPen\WObj:=wPaper;
    MoveL Offs(pOrigin,196.58,177.02,6.00),vTravel,z5,tPen\WObj:=wPaper;
    MoveL Offs(pOrigin,196.58,177.02,0.00),v60,z0,tPen\WObj:=wPaper;
    MoveL Offs(pOrigin,194.47,179.13,0.00),v40,z0,tPen\WObj:=wPaper;
    MoveL Offs(pOrigin,195.18,178.82,0.00),v40,z0,tPen\WObj:=wPaper;
    MoveL Offs(pOrigin,195.60,179.04,0.00),v40,z0,tPen\WObj:=wPaper;
    MoveL Offs(pOrigin,195.18,178.82,0.00),v40,z0,tPen\WObj:=wPaper;
    MoveL Offs(pOrigin,195.52,179.57,0.00),v40,z0,tPen\WObj:=wPaper;
    MoveL Offs(pOrigin,197.62,177.47,0.00),v40,z0,tPen\WObj:=wPaper;
    MoveL Offs(pOrigin,198.52,178.07,0.00),v40,z0,tPen\WObj:=wPaper;
    MoveL Offs(pOrigin,196.27,180.32,0.00),v40,fine,tPen\WObj:=wPaper;
    MoveL Offs(pOrigin,196.27,180.32,6.00),v60,z5,tPen\WObj:=wPaper;
    MoveL Offs(pOrigin,200.31,182.26,6.00),vTravel,z5,tPen\WObj:=wPaper;
    MoveL Offs(pOrigin,200.31,182.26,0.00),v60,z0,tPen\WObj:=wPaper;
    MoveL Offs(pOrigin,202.56,180.00,0.00),v40,z0,tPen\WObj:=wPaper;
    MoveL Offs(pOrigin,203.46,180.60,0.00),v40,z0,tPen\WObj:=wPaper;
    MoveL Offs(pOrigin,201.20,182.85,0.00),v40,z0,tPen\WObj:=wPaper;
    MoveL Offs(pOrigin,200.91,181.80,0.00),v40,z0,tPen\WObj:=wPaper;
    MoveL Offs(pOrigin,201.34,182.01,0.00),v40,z0,tPen\WObj:=wPaper;
    MoveL Offs(pOrigin,200.91,181.80,0.00),v40,fine,tPen\WObj:=wPaper;
    MoveL Offs(pOrigin,200.91,181.80,6.00),v60,z5,tPen\WObj:=wPaper;
    MoveL Offs(pOrigin,202.25,183.30,6.00),vTravel,z5,tPen\WObj:=wPaper;
    MoveL Offs(pOrigin,202.25,183.30,0.00),v60,z0,tPen\WObj:=wPaper;
    MoveL Offs(pOrigin,204.50,181.04,0.00),v40,z0,tPen\WObj:=wPaper;
    MoveL Offs(pOrigin,203.68,181.80,0.00),v40,z0,tPen\WObj:=wPaper;
    MoveL Offs(pOrigin,204.10,182.01,0.00),v40,z0,tPen\WObj:=wPaper;
    MoveL Offs(pOrigin,203.68,181.80,0.00),v40,fine,tPen\WObj:=wPaper;
    MoveL Offs(pOrigin,203.68,181.80,6.00),v60,z5,tPen\WObj:=wPaper;
    MoveL Offs(pOrigin,204.52,183.71,6.00),vTravel,z5,tPen\WObj:=wPaper;
    MoveL Offs(pOrigin,204.52,183.71,0.00),v60,z0,tPen\WObj:=wPaper;
    MoveL Offs(pOrigin,204.95,183.93,0.00),v40,z0,tPen\WObj:=wPaper;
    MoveL Offs(pOrigin,204.52,183.71,0.00),v40,z0,tPen\WObj:=wPaper;
    MoveL Offs(pOrigin,205.59,183.96,0.00),v40,z0,tPen\WObj:=wPaper;
    MoveL Offs(pOrigin,207.92,183.96,0.00),v40,z0,tPen\WObj:=wPaper;
    MoveL Offs(pOrigin,207.50,183.93,0.00),v40,z0,tPen\WObj:=wPaper;
    MoveL Offs(pOrigin,207.93,184.14,0.00),v40,z0,tPen\WObj:=wPaper;
    MoveL Offs(pOrigin,207.50,183.93,0.00),v40,z0,tPen\WObj:=wPaper;
    MoveL Offs(pOrigin,208.35,184.35,0.00),v40,z0,tPen\WObj:=wPaper;
    MoveL Offs(pOrigin,208.77,184.56,0.00),v40,z0,tPen\WObj:=wPaper;
    MoveL Offs(pOrigin,208.35,184.35,0.00),v40,z0,tPen\WObj:=wPaper;
    MoveL Offs(pOrigin,208.24,183.28,0.00),v40,z0,tPen\WObj:=wPaper;
    MoveL Offs(pOrigin,202.53,188.99,0.00),v40,z0,tPen\WObj:=wPaper;
    MoveL Offs(pOrigin,203.07,188.43,0.00),v40,z0,tPen\WObj:=wPaper;
    MoveL Offs(pOrigin,201.41,186.77,0.00),v40,z0,tPen\WObj:=wPaper;
    MoveL Offs(pOrigin,200.74,186.30,0.00),v40,z0,tPen\WObj:=wPaper;
    MoveL Offs(pOrigin,194.13,192.91,0.00),v40,z0,tPen\WObj:=wPaper;
    MoveL Offs(pOrigin,193.39,192.16,0.00),v40,z0,tPen\WObj:=wPaper;
    MoveL Offs(pOrigin,194.74,190.81,0.00),v40,z0,tPen\WObj:=wPaper;
    MoveL Offs(pOrigin,193.99,190.06,0.00),v40,z0,tPen\WObj:=wPaper;
    MoveL Offs(pOrigin,192.64,191.42,0.00),v40,z0,tPen\WObj:=wPaper;
    MoveL Offs(pOrigin,192.04,190.52,0.00),v40,z0,tPen\WObj:=wPaper;
    MoveL Offs(pOrigin,193.39,189.17,0.00),v40,z0,tPen\WObj:=wPaper;
    MoveL Offs(pOrigin,192.95,188.12,0.00),v40,z0,tPen\WObj:=wPaper;
    MoveL Offs(pOrigin,191.45,189.62,0.00),v40,z0,tPen\WObj:=wPaper;
    MoveL Offs(pOrigin,191.00,188.58,0.00),v40,z0,tPen\WObj:=wPaper;
    MoveL Offs(pOrigin,192.35,187.22,0.00),v40,z0,tPen\WObj:=wPaper;
    MoveL Offs(pOrigin,192.28,188.09,0.00),v40,z0,tPen\WObj:=wPaper;
    MoveL Offs(pOrigin,190.18,185.99,0.00),v40,z0,tPen\WObj:=wPaper;
    MoveL Offs(pOrigin,189.96,186.63,0.00),v40,z0,tPen\WObj:=wPaper;
    MoveL Offs(pOrigin,191.46,185.13,0.00),v40,z0,tPen\WObj:=wPaper;
    MoveL Offs(pOrigin,190.92,185.24,0.00),v40,z0,tPen\WObj:=wPaper;
    MoveL Offs(pOrigin,189.42,183.74,0.00),v40,z0,tPen\WObj:=wPaper;
    MoveL Offs(pOrigin,189.86,183.50,0.00),v40,z0,tPen\WObj:=wPaper;
    MoveL Offs(pOrigin,190.07,182.65,0.00),v40,z0,tPen\WObj:=wPaper;
    MoveL Offs(pOrigin,189.86,182.44,0.00),v40,z0,tPen\WObj:=wPaper;
    MoveL Offs(pOrigin,189.86,182.44,0.00),v40,z0,tPen\WObj:=wPaper;
    MoveL Offs(pOrigin,189.86,181.80,0.00),v40,z0,tPen\WObj:=wPaper;
    MoveL Offs(pOrigin,189.23,181.38,0.00),v40,z0,tPen\WObj:=wPaper;
    MoveL Offs(pOrigin,188.66,181.49,0.00),v40,z0,tPen\WObj:=wPaper;
    MoveL Offs(pOrigin,190.02,182.84,0.00),v40,z0,tPen\WObj:=wPaper;
    MoveL Offs(pOrigin,190.72,182.88,0.00),v40,z0,tPen\WObj:=wPaper;
    MoveL Offs(pOrigin,189.06,184.54,0.00),v40,z0,tPen\WObj:=wPaper;
    MoveL Offs(pOrigin,188.62,183.49,0.00),v40,z0,tPen\WObj:=wPaper;
    MoveL Offs(pOrigin,190.42,181.69,0.00),v40,fine,tPen\WObj:=wPaper;
    MoveL Offs(pOrigin,190.42,181.69,6.00),v60,z5,tPen\WObj:=wPaper;
    MoveL Offs(pOrigin,190.28,180.34,6.00),vTravel,z5,tPen\WObj:=wPaper;
    MoveL Offs(pOrigin,190.28,180.34,0.00),v60,z0,tPen\WObj:=wPaper;
    MoveL Offs(pOrigin,188.32,182.29,0.00),v40,fine,tPen\WObj:=wPaper;
    MoveL Offs(pOrigin,188.32,182.29,6.00),v60,z5,tPen\WObj:=wPaper;
    MoveL Offs(pOrigin,188.03,181.09,6.00),vTravel,z5,tPen\WObj:=wPaper;
    MoveL Offs(pOrigin,188.03,181.09,0.00),v60,z0,tPen\WObj:=wPaper;
    MoveL Offs(pOrigin,189.98,179.14,0.00),v40,z0,tPen\WObj:=wPaper;
    MoveL Offs(pOrigin,189.41,179.25,0.00),v40,z0,tPen\WObj:=wPaper;
    MoveL Offs(pOrigin,188.35,178.19,0.00),v40,z0,tPen\WObj:=wPaper;
    MoveL Offs(pOrigin,187.59,178.55,0.00),v40,z0,tPen\WObj:=wPaper;
    MoveL Offs(pOrigin,189.69,176.45,0.00),v40,fine,tPen\WObj:=wPaper;
    MoveL Offs(pOrigin,189.69,176.45,6.00),v60,z5,tPen\WObj:=wPaper;
    MoveL Offs(pOrigin,189.69,174.95,6.00),vTravel,z5,tPen\WObj:=wPaper;
    MoveL Offs(pOrigin,189.69,174.95,0.00),v60,z0,tPen\WObj:=wPaper;
    MoveL Offs(pOrigin,187.59,177.05,0.00),v40,fine,tPen\WObj:=wPaper;
    MoveL Offs(pOrigin,187.59,177.05,6.00),v60,z5,tPen\WObj:=wPaper;
    MoveL Offs(pOrigin,187.44,175.70,6.00),vTravel,z5,tPen\WObj:=wPaper;
    MoveL Offs(pOrigin,187.44,175.70,0.00),v60,z0,tPen\WObj:=wPaper;
    MoveL Offs(pOrigin,189.70,173.45,0.00),v40,fine,tPen\WObj:=wPaper;
    MoveL Offs(pOrigin,189.70,173.45,6.00),v60,z5,tPen\WObj:=wPaper;
    MoveL Offs(pOrigin,189.70,171.95,6.00),vTravel,z5,tPen\WObj:=wPaper;
    MoveL Offs(pOrigin,189.70,171.95,0.00),v60,z0,tPen\WObj:=wPaper;
    MoveL Offs(pOrigin,187.45,174.21,0.00),v40,fine,tPen\WObj:=wPaper;
    MoveL Offs(pOrigin,187.45,174.21,6.00),v60,z5,tPen\WObj:=wPaper;
    MoveL Offs(pOrigin,187.45,172.71,6.00),vTravel,z5,tPen\WObj:=wPaper;
    MoveL Offs(pOrigin,187.45,172.71,0.00),v60,z0,tPen\WObj:=wPaper;
  ENDPROC

  PROC DrawPart162()
    MoveL Offs(pOrigin,189.71,170.45,0.00),v40,fine,tPen\WObj:=wPaper;
    MoveL Offs(pOrigin,189.71,170.45,6.00),v60,z5,tPen\WObj:=wPaper;
    MoveL Offs(pOrigin,191.01,184.08,6.00),vTravel,z5,tPen\WObj:=wPaper;
    MoveL Offs(pOrigin,191.01,184.08,0.00),v60,z0,tPen\WObj:=wPaper;
    MoveL Offs(pOrigin,189.51,185.58,0.00),v40,fine,tPen\WObj:=wPaper;
    MoveL Offs(pOrigin,189.51,185.58,6.00),v60,z5,tPen\WObj:=wPaper;
    MoveL Offs(pOrigin,190.40,187.68,6.00),vTravel,z5,tPen\WObj:=wPaper;
    MoveL Offs(pOrigin,190.40,187.68,0.00),v60,z0,tPen\WObj:=wPaper;
    MoveL Offs(pOrigin,191.91,186.18,0.00),v40,fine,tPen\WObj:=wPaper;
    MoveL Offs(pOrigin,191.91,186.18,6.00),v60,z5,tPen\WObj:=wPaper;
    MoveL Offs(pOrigin,195.64,189.91,6.00),vTravel,z5,tPen\WObj:=wPaper;
    MoveL Offs(pOrigin,195.64,189.91,0.00),v60,z0,tPen\WObj:=wPaper;
    MoveL Offs(pOrigin,198.34,187.20,0.00),v40,z0,tPen\WObj:=wPaper;
    MoveL Offs(pOrigin,199.17,187.51,0.00),v40,z0,tPen\WObj:=wPaper;
    MoveL Offs(pOrigin,200.82,189.17,0.00),v40,fine,tPen\WObj:=wPaper;
    MoveL Offs(pOrigin,200.82,189.17,6.00),v60,z5,tPen\WObj:=wPaper;
    MoveL Offs(pOrigin,200.28,191.24,6.00),vTravel,z5,tPen\WObj:=wPaper;
    MoveL Offs(pOrigin,200.28,191.24,0.00),v60,z0,tPen\WObj:=wPaper;
    MoveL Offs(pOrigin,198.18,193.35,0.00),v40,z0,tPen\WObj:=wPaper;
    MoveL Offs(pOrigin,199.00,193.27,0.00),v40,z0,tPen\WObj:=wPaper;
    MoveL Offs(pOrigin,199.64,193.91,0.00),v40,z0,tPen\WObj:=wPaper;
    MoveL Offs(pOrigin,199.00,193.27,0.00),v40,z0,tPen\WObj:=wPaper;
    MoveL Offs(pOrigin,199.64,193.46,0.00),v40,z0,tPen\WObj:=wPaper;
    MoveL Offs(pOrigin,200.91,193.46,0.00),v40,z0,tPen\WObj:=wPaper;
    MoveL Offs(pOrigin,201.34,193.49,0.00),v40,z0,tPen\WObj:=wPaper;
    MoveL Offs(pOrigin,202.40,194.76,0.00),v40,z0,tPen\WObj:=wPaper;
    MoveL Offs(pOrigin,201.34,193.49,0.00),v40,z0,tPen\WObj:=wPaper;
    MoveL Offs(pOrigin,201.62,192.89,0.00),v40,z0,tPen\WObj:=wPaper;
    MoveL Offs(pOrigin,197.72,196.79,0.00),v40,z0,tPen\WObj:=wPaper;
    MoveL Offs(pOrigin,197.12,195.90,0.00),v40,z0,tPen\WObj:=wPaper;
    MoveL Offs(pOrigin,198.02,195.00,0.00),v40,z0,tPen\WObj:=wPaper;
    MoveL Offs(pOrigin,198.77,194.24,0.00),v40,z0,tPen\WObj:=wPaper;
    MoveL Offs(pOrigin,201.03,191.99,0.00),v40,z0,tPen\WObj:=wPaper;
    MoveL Offs(pOrigin,200.27,192.43,0.00),v40,z0,tPen\WObj:=wPaper;
    MoveL Offs(pOrigin,200.70,192.85,0.00),v40,z0,tPen\WObj:=wPaper;
    MoveL Offs(pOrigin,200.27,192.43,0.00),v40,z0,tPen\WObj:=wPaper;
    MoveL Offs(pOrigin,200.06,192.41,0.00),v40,z0,tPen\WObj:=wPaper;
    MoveL Offs(pOrigin,198.58,192.41,0.00),v40,z0,tPen\WObj:=wPaper;
    MoveL Offs(pOrigin,197.94,192.00,0.00),v40,z0,tPen\WObj:=wPaper;
    MoveL Offs(pOrigin,198.79,192.85,0.00),v40,z0,tPen\WObj:=wPaper;
    MoveL Offs(pOrigin,197.94,192.00,0.00),v40,z0,tPen\WObj:=wPaper;
    MoveL Offs(pOrigin,197.73,191.35,0.00),v40,z0,tPen\WObj:=wPaper;
    MoveL Offs(pOrigin,199.21,191.35,0.00),v40,z0,tPen\WObj:=wPaper;
    MoveL Offs(pOrigin,199.85,191.79,0.00),v40,z0,tPen\WObj:=wPaper;
    MoveL Offs(pOrigin,200.06,192.21,0.00),v40,z0,tPen\WObj:=wPaper;
    MoveL Offs(pOrigin,199.85,191.79,0.00),v40,fine,tPen\WObj:=wPaper;
    MoveL Offs(pOrigin,199.85,191.79,6.00),v60,z5,tPen\WObj:=wPaper;
    MoveL Offs(pOrigin,197.43,192.60,6.00),vTravel,z5,tPen\WObj:=wPaper;
    MoveL Offs(pOrigin,197.43,192.60,0.00),v60,z0,tPen\WObj:=wPaper;
    MoveL Offs(pOrigin,207.35,182.68,0.00),v40,z0,tPen\WObj:=wPaper;
    MoveL Offs(pOrigin,206.30,182.24,0.00),v40,z0,tPen\WObj:=wPaper;
    MoveL Offs(pOrigin,194.73,193.81,0.00),v40,z0,tPen\WObj:=wPaper;
    MoveL Offs(pOrigin,195.63,194.40,0.00),v40,z0,tPen\WObj:=wPaper;
    MoveL Offs(pOrigin,196.53,193.50,0.00),v40,z0,tPen\WObj:=wPaper;
    MoveL Offs(pOrigin,197.12,194.40,0.00),v40,z0,tPen\WObj:=wPaper;
    MoveL Offs(pOrigin,196.22,195.30,0.00),v40,fine,tPen\WObj:=wPaper;
    MoveL Offs(pOrigin,196.22,195.30,6.00),v60,z5,tPen\WObj:=wPaper;
    MoveL Offs(pOrigin,198.61,197.39,6.00),vTravel,z5,tPen\WObj:=wPaper;
    MoveL Offs(pOrigin,198.61,197.39,0.00),v60,z0,tPen\WObj:=wPaper;
    MoveL Offs(pOrigin,202.22,193.78,0.00),v40,z0,tPen\WObj:=wPaper;
    MoveL Offs(pOrigin,201.98,194.52,0.00),v40,z0,tPen\WObj:=wPaper;
    MoveL Offs(pOrigin,200.28,194.52,0.00),v40,z0,tPen\WObj:=wPaper;
    MoveL Offs(pOrigin,200.27,194.76,0.00),v40,z0,tPen\WObj:=wPaper;
    MoveL Offs(pOrigin,200.91,195.40,0.00),v40,z0,tPen\WObj:=wPaper;
    MoveL Offs(pOrigin,200.27,194.76,0.00),v40,fine,tPen\WObj:=wPaper;
    MoveL Offs(pOrigin,200.27,194.76,6.00),v60,z5,tPen\WObj:=wPaper;
    MoveL Offs(pOrigin,201.34,195.58,6.00),vTravel,z5,tPen\WObj:=wPaper;
    MoveL Offs(pOrigin,201.34,195.58,0.00),v60,z0,tPen\WObj:=wPaper;
    MoveL Offs(pOrigin,202.82,195.58,0.00),v40,z0,tPen\WObj:=wPaper;
    MoveL Offs(pOrigin,203.71,195.28,0.00),v40,z0,tPen\WObj:=wPaper;
    MoveL Offs(pOrigin,200.41,198.58,0.00),v40,z0,tPen\WObj:=wPaper;
    MoveL Offs(pOrigin,199.51,197.99,0.00),v40,z0,tPen\WObj:=wPaper;
    MoveL Offs(pOrigin,203.12,194.38,0.00),v40,fine,tPen\WObj:=wPaper;
    MoveL Offs(pOrigin,203.12,194.38,6.00),v60,z5,tPen\WObj:=wPaper;
    MoveL Offs(pOrigin,203.68,196.63,6.00),vTravel,z5,tPen\WObj:=wPaper;
    MoveL Offs(pOrigin,203.68,196.63,0.00),v60,z0,tPen\WObj:=wPaper;
    MoveL Offs(pOrigin,202.19,196.63,0.00),v40,z0,tPen\WObj:=wPaper;
    MoveL Offs(pOrigin,202.19,197.10,0.00),v40,z0,tPen\WObj:=wPaper;
    MoveL Offs(pOrigin,203.25,198.16,0.00),v40,z0,tPen\WObj:=wPaper;
    MoveL Offs(pOrigin,202.19,197.10,0.00),v40,z0,tPen\WObj:=wPaper;
    MoveL Offs(pOrigin,201.55,196.25,0.00),v40,z0,tPen\WObj:=wPaper;
    MoveL Offs(pOrigin,201.98,196.68,0.00),v40,z0,tPen\WObj:=wPaper;
    MoveL Offs(pOrigin,201.55,196.25,0.00),v40,fine,tPen\WObj:=wPaper;
    MoveL Offs(pOrigin,201.55,196.25,6.00),v60,z5,tPen\WObj:=wPaper;
    MoveL Offs(pOrigin,203.55,199.92,6.00),vTravel,z5,tPen\WObj:=wPaper;
    MoveL Offs(pOrigin,203.55,199.92,0.00),v60,z0,tPen\WObj:=wPaper;
    MoveL Offs(pOrigin,205.80,197.67,0.00),v40,z0,tPen\WObj:=wPaper;
    MoveL Offs(pOrigin,206.40,198.56,0.00),v40,z0,tPen\WObj:=wPaper;
    MoveL Offs(pOrigin,204.29,200.67,0.00),v40,z0,tPen\WObj:=wPaper;
    MoveL Offs(pOrigin,204.95,200.29,0.00),v40,z0,tPen\WObj:=wPaper;
    MoveL Offs(pOrigin,205.38,200.71,0.00),v40,z0,tPen\WObj:=wPaper;
    MoveL Offs(pOrigin,204.95,200.29,0.00),v40,z0,tPen\WObj:=wPaper;
    MoveL Offs(pOrigin,204.95,199.80,0.00),v40,z0,tPen\WObj:=wPaper;
    MoveL Offs(pOrigin,206.44,199.80,0.00),v40,z0,tPen\WObj:=wPaper;
    MoveL Offs(pOrigin,207.15,199.31,0.00),v40,z0,tPen\WObj:=wPaper;
    MoveL Offs(pOrigin,204.89,201.57,0.00),v40,z0,tPen\WObj:=wPaper;
    MoveL Offs(pOrigin,205.80,201.35,0.00),v40,z0,tPen\WObj:=wPaper;
    MoveL Offs(pOrigin,206.23,201.77,0.00),v40,z0,tPen\WObj:=wPaper;
    MoveL Offs(pOrigin,205.80,201.35,0.00),v40,z0,tPen\WObj:=wPaper;
    MoveL Offs(pOrigin,205.80,200.86,0.00),v40,z0,tPen\WObj:=wPaper;
    MoveL Offs(pOrigin,207.29,200.86,0.00),v40,z0,tPen\WObj:=wPaper;
    MoveL Offs(pOrigin,207.45,200.27,0.00),v40,z0,tPen\WObj:=wPaper;
    MoveL Offs(pOrigin,196.33,189.15,0.00),v40,z0,tPen\WObj:=wPaper;
    MoveL Offs(pOrigin,197.49,189.24,0.00),v40,z0,tPen\WObj:=wPaper;
    MoveL Offs(pOrigin,197.49,190.30,0.00),v40,fine,tPen\WObj:=wPaper;
    MoveL Offs(pOrigin,197.49,190.30,6.00),v60,z5,tPen\WObj:=wPaper;
    MoveL Offs(pOrigin,205.59,182.86,6.00),vTravel,z5,tPen\WObj:=wPaper;
    MoveL Offs(pOrigin,205.59,182.86,0.00),v60,z0,tPen\WObj:=wPaper;
    MoveL Offs(pOrigin,206.01,183.07,0.00),v40,z0,tPen\WObj:=wPaper;
    MoveL Offs(pOrigin,205.59,182.86,0.00),v40,fine,tPen\WObj:=wPaper;
    MoveL Offs(pOrigin,205.59,182.86,6.00),v60,z5,tPen\WObj:=wPaper;
    MoveL Offs(pOrigin,209.41,186.26,6.00),vTravel,z5,tPen\WObj:=wPaper;
    MoveL Offs(pOrigin,209.41,186.26,0.00),v60,z0,tPen\WObj:=wPaper;
    MoveL Offs(pOrigin,209.84,186.48,0.00),v40,z0,tPen\WObj:=wPaper;
    MoveL Offs(pOrigin,209.41,186.26,0.00),v40,z0,tPen\WObj:=wPaper;
    MoveL Offs(pOrigin,210.05,186.69,0.00),v40,z0,tPen\WObj:=wPaper;
    MoveL Offs(pOrigin,210.69,187.11,0.00),v40,z0,tPen\WObj:=wPaper;
    MoveL Offs(pOrigin,210.05,186.69,0.00),v40,z0,tPen\WObj:=wPaper;
    MoveL Offs(pOrigin,209.88,187.62,0.00),v40,z0,tPen\WObj:=wPaper;
    MoveL Offs(pOrigin,211.83,185.67,0.00),v40,z0,tPen\WObj:=wPaper;
  ENDPROC

  PROC DrawPart163()
    MoveL Offs(pOrigin,212.73,186.26,0.00),v40,z0,tPen\WObj:=wPaper;
    MoveL Offs(pOrigin,210.92,188.06,0.00),v40,fine,tPen\WObj:=wPaper;
    MoveL Offs(pOrigin,210.92,188.06,6.00),v60,z5,tPen\WObj:=wPaper;
    MoveL Offs(pOrigin,208.98,187.02,6.00),vTravel,z5,tPen\WObj:=wPaper;
    MoveL Offs(pOrigin,208.98,187.02,0.00),v60,z0,tPen\WObj:=wPaper;
    MoveL Offs(pOrigin,210.93,185.07,0.00),v40,fine,tPen\WObj:=wPaper;
    MoveL Offs(pOrigin,210.93,185.07,6.00),v60,z5,tPen\WObj:=wPaper;
    MoveL Offs(pOrigin,215.12,188.35,6.00),vTravel,z5,tPen\WObj:=wPaper;
    MoveL Offs(pOrigin,215.12,188.35,0.00),v60,z0,tPen\WObj:=wPaper;
    MoveL Offs(pOrigin,213.47,190.00,0.00),v40,z0,tPen\WObj:=wPaper;
    MoveL Offs(pOrigin,214.21,190.75,0.00),v40,z0,tPen\WObj:=wPaper;
    MoveL Offs(pOrigin,216.02,188.95,0.00),v40,z0,tPen\WObj:=wPaper;
    MoveL Offs(pOrigin,216.91,189.54,0.00),v40,z0,tPen\WObj:=wPaper;
    MoveL Offs(pOrigin,215.11,191.35,0.00),v40,z0,tPen\WObj:=wPaper;
    MoveL Offs(pOrigin,216.01,191.94,0.00),v40,z0,tPen\WObj:=wPaper;
    MoveL Offs(pOrigin,217.66,190.29,0.00),v40,z0,tPen\WObj:=wPaper;
    MoveL Offs(pOrigin,218.41,191.04,0.00),v40,z0,tPen\WObj:=wPaper;
    MoveL Offs(pOrigin,216.60,192.84,0.00),v40,z0,tPen\WObj:=wPaper;
    MoveL Offs(pOrigin,217.50,193.44,0.00),v40,z0,tPen\WObj:=wPaper;
    MoveL Offs(pOrigin,219.15,191.78,0.00),v40,z0,tPen\WObj:=wPaper;
    MoveL Offs(pOrigin,219.90,192.53,0.00),v40,z0,tPen\WObj:=wPaper;
    MoveL Offs(pOrigin,218.25,194.18,0.00),v40,z0,tPen\WObj:=wPaper;
    MoveL Offs(pOrigin,218.99,194.93,0.00),v40,z0,tPen\WObj:=wPaper;
    MoveL Offs(pOrigin,220.80,193.13,0.00),v40,z0,tPen\WObj:=wPaper;
    MoveL Offs(pOrigin,220.76,194.17,0.00),v40,z0,tPen\WObj:=wPaper;
    MoveL Offs(pOrigin,223.31,196.73,0.00),v40,z0,tPen\WObj:=wPaper;
    MoveL Offs(pOrigin,223.01,196.63,0.00),v40,z0,tPen\WObj:=wPaper;
    MoveL Offs(pOrigin,221.74,196.63,0.00),v40,fine,tPen\WObj:=wPaper;
    MoveL Offs(pOrigin,221.74,196.63,6.00),v60,z5,tPen\WObj:=wPaper;
    MoveL Offs(pOrigin,220.49,196.42,6.00),vTravel,z5,tPen\WObj:=wPaper;
    MoveL Offs(pOrigin,220.49,196.42,0.00),v60,z0,tPen\WObj:=wPaper;
    MoveL Offs(pOrigin,225.29,191.62,0.00),v40,z0,tPen\WObj:=wPaper;
    MoveL Offs(pOrigin,224.29,191.35,0.00),v40,z0,tPen\WObj:=wPaper;
    MoveL Offs(pOrigin,223.01,191.35,0.00),v40,z0,tPen\WObj:=wPaper;
    MoveL Offs(pOrigin,222.40,191.33,0.00),v40,z0,tPen\WObj:=wPaper;
    MoveL Offs(pOrigin,224.20,193.13,0.00),v40,z0,tPen\WObj:=wPaper;
    MoveL Offs(pOrigin,223.65,193.46,0.00),v40,z0,tPen\WObj:=wPaper;
    MoveL Offs(pOrigin,222.59,193.46,0.00),v40,fine,tPen\WObj:=wPaper;
    MoveL Offs(pOrigin,222.59,193.46,6.00),v60,z5,tPen\WObj:=wPaper;
    MoveL Offs(pOrigin,221.85,192.08,6.00),vTravel,z5,tPen\WObj:=wPaper;
    MoveL Offs(pOrigin,221.85,192.08,0.00),v60,z0,tPen\WObj:=wPaper;
    MoveL Offs(pOrigin,225.90,188.02,0.00),v40,z0,tPen\WObj:=wPaper;
    MoveL Offs(pOrigin,225.68,187.15,0.00),v40,z0,tPen\WObj:=wPaper;
    MoveL Offs(pOrigin,223.88,185.34,0.00),v40,z0,tPen\WObj:=wPaper;
    MoveL Offs(pOrigin,224.50,185.02,0.00),v40,z0,tPen\WObj:=wPaper;
    MoveL Offs(pOrigin,225.56,185.02,0.00),v40,z0,tPen\WObj:=wPaper;
    MoveL Offs(pOrigin,226.12,184.60,0.00),v40,z0,tPen\WObj:=wPaper;
    MoveL Offs(pOrigin,224.32,182.80,0.00),v40,z0,tPen\WObj:=wPaper;
    MoveL Offs(pOrigin,223.82,182.63,0.00),v40,z0,tPen\WObj:=wPaper;
    MoveL Offs(pOrigin,230.44,176.02,0.00),v40,z0,tPen\WObj:=wPaper;
    MoveL Offs(pOrigin,229.99,176.52,0.00),v40,z0,tPen\WObj:=wPaper;
    MoveL Offs(pOrigin,225.94,172.47,0.00),v40,z0,tPen\WObj:=wPaper;
    MoveL Offs(pOrigin,226.41,172.34,0.00),v40,z0,tPen\WObj:=wPaper;
    MoveL Offs(pOrigin,228.75,172.34,0.00),v40,z0,tPen\WObj:=wPaper;
    MoveL Offs(pOrigin,228.96,173.40,0.00),v40,z0,tPen\WObj:=wPaper;
    MoveL Offs(pOrigin,226.41,173.40,0.00),v40,z0,tPen\WObj:=wPaper;
    MoveL Offs(pOrigin,225.79,173.81,0.00),v40,z0,tPen\WObj:=wPaper;
    MoveL Offs(pOrigin,230.75,178.77,0.00),v40,z0,tPen\WObj:=wPaper;
    MoveL Offs(pOrigin,230.88,178.82,0.00),v40,z0,tPen\WObj:=wPaper;
    MoveL Offs(pOrigin,230.31,179.25,0.00),v40,z0,tPen\WObj:=wPaper;
    MoveL Offs(pOrigin,229.81,180.52,0.00),v40,z0,tPen\WObj:=wPaper;
    MoveL Offs(pOrigin,229.81,182.65,0.00),v40,z0,tPen\WObj:=wPaper;
    MoveL Offs(pOrigin,230.38,185.62,0.00),v40,z0,tPen\WObj:=wPaper;
    MoveL Offs(pOrigin,231.73,187.18,0.00),v40,z0,tPen\WObj:=wPaper;
    MoveL Offs(pOrigin,233.85,187.32,0.00),v40,z0,tPen\WObj:=wPaper;
    MoveL Offs(pOrigin,233.85,187.32,0.00),v40,z0,tPen\WObj:=wPaper;
    MoveL Offs(pOrigin,233.57,188.10,0.00),v40,z0,tPen\WObj:=wPaper;
    MoveL Offs(pOrigin,231.94,188.39,0.00),v40,z0,tPen\WObj:=wPaper;
    MoveL Offs(pOrigin,230.66,187.75,0.00),v40,z0,tPen\WObj:=wPaper;
    MoveL Offs(pOrigin,229.53,186.48,0.00),v40,z0,tPen\WObj:=wPaper;
    MoveL Offs(pOrigin,228.75,183.71,0.00),v40,z0,tPen\WObj:=wPaper;
    MoveL Offs(pOrigin,228.32,176.49,0.00),v40,z0,tPen\WObj:=wPaper;
    MoveL Offs(pOrigin,228.04,175.43,0.00),v40,z0,tPen\WObj:=wPaper;
    MoveL Offs(pOrigin,227.69,175.21,0.00),v40,z0,tPen\WObj:=wPaper;
    MoveL Offs(pOrigin,227.69,175.21,0.00),v40,z0,tPen\WObj:=wPaper;
    MoveL Offs(pOrigin,227.26,175.85,0.00),v40,z0,tPen\WObj:=wPaper;
    MoveL Offs(pOrigin,227.05,178.40,0.00),v40,z0,tPen\WObj:=wPaper;
    MoveL Offs(pOrigin,224.93,189.24,0.00),v40,z0,tPen\WObj:=wPaper;
    MoveL Offs(pOrigin,222.16,201.14,0.00),v40,z0,tPen\WObj:=wPaper;
    MoveL Offs(pOrigin,221.10,207.30,0.00),v40,z0,tPen\WObj:=wPaper;
    MoveL Offs(pOrigin,221.31,208.57,0.00),v40,z0,tPen\WObj:=wPaper;
    MoveL Offs(pOrigin,222.16,208.15,0.00),v40,z0,tPen\WObj:=wPaper;
    MoveL Offs(pOrigin,224.93,205.39,0.00),v40,z0,tPen\WObj:=wPaper;
    MoveL Offs(pOrigin,230.80,195.40,0.00),v40,z0,tPen\WObj:=wPaper;
    MoveL Offs(pOrigin,239.23,183.29,0.00),v40,z0,tPen\WObj:=wPaper;
    MoveL Offs(pOrigin,241.36,179.25,0.00),v40,z0,tPen\WObj:=wPaper;
    MoveL Offs(pOrigin,243.98,171.60,0.00),v40,z0,tPen\WObj:=wPaper;
    MoveL Offs(pOrigin,245.11,169.48,0.00),v40,z0,tPen\WObj:=wPaper;
    MoveL Offs(pOrigin,251.91,163.95,0.00),v40,z0,tPen\WObj:=wPaper;
    MoveL Offs(pOrigin,251.70,162.68,0.00),v40,z0,tPen\WObj:=wPaper;
    MoveL Offs(pOrigin,249.36,160.12,0.00),v40,z0,tPen\WObj:=wPaper;
    MoveL Offs(pOrigin,247.52,157.36,0.00),v40,z0,tPen\WObj:=wPaper;
    MoveL Offs(pOrigin,245.96,152.69,0.00),v40,z0,tPen\WObj:=wPaper;
    MoveL Offs(pOrigin,245.65,153.35,0.00),v40,z0,tPen\WObj:=wPaper;
    MoveL Offs(pOrigin,247.76,155.46,0.00),v40,z0,tPen\WObj:=wPaper;
    MoveL Offs(pOrigin,248.48,154.99,0.00),v40,z0,tPen\WObj:=wPaper;
    MoveL Offs(pOrigin,246.37,157.10,0.00),v40,z0,tPen\WObj:=wPaper;
    MoveL Offs(pOrigin,246.86,157.55,0.00),v40,z0,tPen\WObj:=wPaper;
    MoveL Offs(pOrigin,260.99,171.68,0.00),v40,z0,tPen\WObj:=wPaper;
    MoveL Offs(pOrigin,261.61,171.73,0.00),v40,z0,tPen\WObj:=wPaper;
    MoveL Offs(pOrigin,259.05,174.29,0.00),v40,z0,tPen\WObj:=wPaper;
    MoveL Offs(pOrigin,259.20,174.37,0.00),v40,z0,tPen\WObj:=wPaper;
    MoveL Offs(pOrigin,266.71,181.88,0.00),v40,z0,tPen\WObj:=wPaper;
    MoveL Offs(pOrigin,266.15,181.85,0.00),v40,z0,tPen\WObj:=wPaper;
    MoveL Offs(pOrigin,264.66,181.85,0.00),v40,z0,tPen\WObj:=wPaper;
    MoveL Offs(pOrigin,263.97,182.81,0.00),v40,z0,tPen\WObj:=wPaper;
    MoveL Offs(pOrigin,267.88,178.90,0.00),v40,z0,tPen\WObj:=wPaper;
    MoveL Offs(pOrigin,267.13,178.16,0.00),v40,z0,tPen\WObj:=wPaper;
    MoveL Offs(pOrigin,263.37,181.91,0.00),v40,z0,tPen\WObj:=wPaper;
    MoveL Offs(pOrigin,263.41,181.57,0.00),v40,z0,tPen\WObj:=wPaper;
    MoveL Offs(pOrigin,272.73,190.89,0.00),v40,z0,tPen\WObj:=wPaper;
    MoveL Offs(pOrigin,272.31,191.35,0.00),v40,z0,tPen\WObj:=wPaper;
    MoveL Offs(pOrigin,271.04,191.35,0.00),v40,z0,tPen\WObj:=wPaper;
    MoveL Offs(pOrigin,269.93,191.78,0.00),v40,z0,tPen\WObj:=wPaper;
    MoveL Offs(pOrigin,283.16,178.56,0.00),v40,z0,tPen\WObj:=wPaper;
    MoveL Offs(pOrigin,282.73,178.48,0.00),v40,z0,tPen\WObj:=wPaper;
    MoveL Offs(pOrigin,279.12,174.88,0.00),v40,z0,tPen\WObj:=wPaper;
    MoveL Offs(pOrigin,279.54,174.46,0.00),v40,z0,tPen\WObj:=wPaper;
    MoveL Offs(pOrigin,281.24,174.46,0.00),v40,z0,tPen\WObj:=wPaper;
    MoveL Offs(pOrigin,281.67,174.44,0.00),v40,z0,tPen\WObj:=wPaper;
  ENDPROC

  PROC DrawPart164()
    MoveL Offs(pOrigin,278.66,171.43,0.00),v40,z0,tPen\WObj:=wPaper;
    MoveL Offs(pOrigin,278.24,171.53,0.00),v40,z0,tPen\WObj:=wPaper;
    MoveL Offs(pOrigin,280.94,168.83,0.00),v40,z0,tPen\WObj:=wPaper;
    MoveL Offs(pOrigin,280.30,168.59,0.00),v40,z0,tPen\WObj:=wPaper;
    MoveL Offs(pOrigin,277.30,165.58,0.00),v40,z0,tPen\WObj:=wPaper;
    MoveL Offs(pOrigin,276.76,165.54,0.00),v40,z0,tPen\WObj:=wPaper;
    MoveL Offs(pOrigin,279.61,162.69,0.00),v40,z0,tPen\WObj:=wPaper;
    MoveL Offs(pOrigin,279.09,162.89,0.00),v40,z0,tPen\WObj:=wPaper;
    MoveL Offs(pOrigin,276.23,160.04,0.00),v40,z0,tPen\WObj:=wPaper;
    MoveL Offs(pOrigin,276.77,159.67,0.00),v40,z0,tPen\WObj:=wPaper;
    MoveL Offs(pOrigin,277.84,159.67,0.00),v40,z0,tPen\WObj:=wPaper;
    MoveL Offs(pOrigin,278.48,159.30,0.00),v40,z0,tPen\WObj:=wPaper;
    MoveL Offs(pOrigin,275.17,155.99,0.00),v40,z0,tPen\WObj:=wPaper;
    MoveL Offs(pOrigin,274.69,155.66,0.00),v40,z0,tPen\WObj:=wPaper;
    MoveL Offs(pOrigin,277.69,152.66,0.00),v40,fine,tPen\WObj:=wPaper;
    MoveL Offs(pOrigin,277.69,152.66,6.00),v60,z5,tPen\WObj:=wPaper;
    MoveL Offs(pOrigin,277.99,153.85,6.00),vTravel,z5,tPen\WObj:=wPaper;
    MoveL Offs(pOrigin,277.99,153.85,0.00),v60,z0,tPen\WObj:=wPaper;
    MoveL Offs(pOrigin,275.13,156.71,0.00),v40,z0,tPen\WObj:=wPaper;
    MoveL Offs(pOrigin,276.14,156.50,0.00),v40,z0,tPen\WObj:=wPaper;
    MoveL Offs(pOrigin,277.41,156.50,0.00),v40,z0,tPen\WObj:=wPaper;
    MoveL Offs(pOrigin,278.43,156.40,0.00),v40,z0,tPen\WObj:=wPaper;
    MoveL Offs(pOrigin,275.58,159.25,0.00),v40,z0,tPen\WObj:=wPaper;
    MoveL Offs(pOrigin,276.56,158.62,0.00),v40,z0,tPen\WObj:=wPaper;
    MoveL Offs(pOrigin,277.62,158.62,0.00),v40,z0,tPen\WObj:=wPaper;
    MoveL Offs(pOrigin,277.62,157.56,0.00),v40,z0,tPen\WObj:=wPaper;
    MoveL Offs(pOrigin,276.35,157.56,0.00),v40,fine,tPen\WObj:=wPaper;
    MoveL Offs(pOrigin,276.35,157.56,6.00),v60,z5,tPen\WObj:=wPaper;
    MoveL Offs(pOrigin,278.02,157.35,6.00),vTravel,z5,tPen\WObj:=wPaper;
    MoveL Offs(pOrigin,278.02,157.35,0.00),v60,z0,tPen\WObj:=wPaper;
    MoveL Offs(pOrigin,274.26,153.59,0.00),v40,z0,tPen\WObj:=wPaper;
    MoveL Offs(pOrigin,273.95,153.42,0.00),v40,z0,tPen\WObj:=wPaper;
    MoveL Offs(pOrigin,277.40,149.96,0.00),v40,z0,tPen\WObj:=wPaper;
    MoveL Offs(pOrigin,276.65,150.00,0.00),v40,z0,tPen\WObj:=wPaper;
    MoveL Offs(pOrigin,273.19,146.55,0.00),v40,fine,tPen\WObj:=wPaper;
    MoveL Offs(pOrigin,273.19,146.55,6.00),v60,z5,tPen\WObj:=wPaper;
    MoveL Offs(pOrigin,274.65,147.00,6.00),vTravel,z5,tPen\WObj:=wPaper;
    MoveL Offs(pOrigin,274.65,147.00,0.00),v60,z0,tPen\WObj:=wPaper;
    MoveL Offs(pOrigin,275.71,147.00,0.00),v40,z0,tPen\WObj:=wPaper;
    MoveL Offs(pOrigin,276.51,146.37,0.00),v40,z0,tPen\WObj:=wPaper;
    MoveL Offs(pOrigin,272.61,150.28,0.00),v40,fine,tPen\WObj:=wPaper;
    MoveL Offs(pOrigin,272.61,150.28,6.00),v60,z5,tPen\WObj:=wPaper;
    MoveL Offs(pOrigin,274.44,150.56,6.00),vTravel,z5,tPen\WObj:=wPaper;
    MoveL Offs(pOrigin,274.44,150.56,0.00),v60,z0,tPen\WObj:=wPaper;
    MoveL Offs(pOrigin,273.73,149.93,0.00),v40,z0,tPen\WObj:=wPaper;
    MoveL Offs(pOrigin,267.78,135.05,0.00),v40,z0,tPen\WObj:=wPaper;
    MoveL Offs(pOrigin,267.64,133.77,0.00),v40,fine,tPen\WObj:=wPaper;
    MoveL Offs(pOrigin,267.64,133.77,6.00),v60,z5,tPen\WObj:=wPaper;
    MoveL Offs(pOrigin,268.76,136.21,6.00),vTravel,z5,tPen\WObj:=wPaper;
    MoveL Offs(pOrigin,268.76,136.21,0.00),v60,z0,tPen\WObj:=wPaper;
    MoveL Offs(pOrigin,268.01,136.96,0.00),v40,z0,tPen\WObj:=wPaper;
    MoveL Offs(pOrigin,268.45,138.01,0.00),v40,z0,tPen\WObj:=wPaper;
    MoveL Offs(pOrigin,269.20,137.25,0.00),v40,z0,tPen\WObj:=wPaper;
    MoveL Offs(pOrigin,269.80,138.15,0.00),v40,z0,tPen\WObj:=wPaper;
    MoveL Offs(pOrigin,268.60,139.35,0.00),v40,z0,tPen\WObj:=wPaper;
    MoveL Offs(pOrigin,269.04,140.40,0.00),v40,z0,tPen\WObj:=wPaper;
    MoveL Offs(pOrigin,270.25,139.20,0.00),v40,z0,tPen\WObj:=wPaper;
    MoveL Offs(pOrigin,270.69,140.25,0.00),v40,z0,tPen\WObj:=wPaper;
    MoveL Offs(pOrigin,269.49,141.45,0.00),v40,z0,tPen\WObj:=wPaper;
    MoveL Offs(pOrigin,269.94,142.49,0.00),v40,z0,tPen\WObj:=wPaper;
    MoveL Offs(pOrigin,271.29,141.14,0.00),v40,fine,tPen\WObj:=wPaper;
    MoveL Offs(pOrigin,271.29,141.14,6.00),v60,z5,tPen\WObj:=wPaper;
    MoveL Offs(pOrigin,271.58,142.34,6.00),vTravel,z5,tPen\WObj:=wPaper;
    MoveL Offs(pOrigin,271.58,142.34,0.00),v60,z0,tPen\WObj:=wPaper;
    MoveL Offs(pOrigin,270.23,143.69,0.00),v40,fine,tPen\WObj:=wPaper;
    MoveL Offs(pOrigin,270.23,143.69,6.00),v60,z5,tPen\WObj:=wPaper;
    MoveL Offs(pOrigin,271.72,148.18,6.00),vTravel,z5,tPen\WObj:=wPaper;
    MoveL Offs(pOrigin,271.72,148.18,0.00),v60,z0,tPen\WObj:=wPaper;
    MoveL Offs(pOrigin,276.07,143.82,0.00),v40,fine,tPen\WObj:=wPaper;
    MoveL Offs(pOrigin,276.07,143.82,6.00),v60,z5,tPen\WObj:=wPaper;
    MoveL Offs(pOrigin,275.92,148.06,6.00),vTravel,z5,tPen\WObj:=wPaper;
    MoveL Offs(pOrigin,275.92,148.06,0.00),v60,z0,tPen\WObj:=wPaper;
    MoveL Offs(pOrigin,274.65,148.06,0.00),v40,z0,tPen\WObj:=wPaper;
    MoveL Offs(pOrigin,274.65,149.11,0.00),v40,z0,tPen\WObj:=wPaper;
    MoveL Offs(pOrigin,276.14,149.11,0.00),v40,z0,tPen\WObj:=wPaper;
    MoveL Offs(pOrigin,277.11,148.76,0.00),v40,z0,tPen\WObj:=wPaper;
    MoveL Offs(pOrigin,273.50,152.37,0.00),v40,fine,tPen\WObj:=wPaper;
    MoveL Offs(pOrigin,273.50,152.37,6.00),v60,z5,tPen\WObj:=wPaper;
    MoveL Offs(pOrigin,274.65,151.22,6.00),vTravel,z5,tPen\WObj:=wPaper;
    MoveL Offs(pOrigin,274.65,151.22,0.00),v60,z0,tPen\WObj:=wPaper;
    MoveL Offs(pOrigin,276.35,151.22,0.00),v40,z0,tPen\WObj:=wPaper;
    MoveL Offs(pOrigin,275.63,151.62,0.00),v40,z0,tPen\WObj:=wPaper;
    MoveL Offs(pOrigin,275.63,153.96,0.00),v40,z0,tPen\WObj:=wPaper;
    MoveL Offs(pOrigin,275.50,154.39,0.00),v40,z0,tPen\WObj:=wPaper;
    MoveL Offs(pOrigin,276.99,154.39,0.00),v40,z0,tPen\WObj:=wPaper;
    MoveL Offs(pOrigin,277.20,155.45,0.00),v40,z0,tPen\WObj:=wPaper;
    MoveL Offs(pOrigin,275.71,155.45,0.00),v40,fine,tPen\WObj:=wPaper;
    MoveL Offs(pOrigin,275.71,155.45,6.00),v60,z5,tPen\WObj:=wPaper;
    MoveL Offs(pOrigin,274.24,154.62,6.00),vTravel,z5,tPen\WObj:=wPaper;
    MoveL Offs(pOrigin,274.24,154.62,0.00),v60,z0,tPen\WObj:=wPaper;
    MoveL Offs(pOrigin,277.55,151.31,0.00),v40,fine,tPen\WObj:=wPaper;
    MoveL Offs(pOrigin,277.55,151.31,6.00),v60,z5,tPen\WObj:=wPaper;
    MoveL Offs(pOrigin,276.14,150.17,6.00),vTravel,z5,tPen\WObj:=wPaper;
    MoveL Offs(pOrigin,276.14,150.17,0.00),v60,z0,tPen\WObj:=wPaper;
    MoveL Offs(pOrigin,274.65,150.17,0.00),v40,fine,tPen\WObj:=wPaper;
    MoveL Offs(pOrigin,274.65,150.17,6.00),v60,z5,tPen\WObj:=wPaper;
    MoveL Offs(pOrigin,278.58,157.75,6.00),vTravel,z5,tPen\WObj:=wPaper;
    MoveL Offs(pOrigin,278.58,157.75,0.00),v60,z0,tPen\WObj:=wPaper;
    MoveL Offs(pOrigin,275.72,160.60,0.00),v40,fine,tPen\WObj:=wPaper;
    MoveL Offs(pOrigin,275.72,160.60,6.00),v60,z5,tPen\WObj:=wPaper;
    MoveL Offs(pOrigin,276.02,161.80,6.00),vTravel,z5,tPen\WObj:=wPaper;
    MoveL Offs(pOrigin,276.02,161.80,0.00),v60,z0,tPen\WObj:=wPaper;
    MoveL Offs(pOrigin,278.87,158.95,0.00),v40,fine,tPen\WObj:=wPaper;
    MoveL Offs(pOrigin,278.87,158.95,6.00),v60,z5,tPen\WObj:=wPaper;
    MoveL Offs(pOrigin,279.02,160.29,6.00),vTravel,z5,tPen\WObj:=wPaper;
    MoveL Offs(pOrigin,279.02,160.29,0.00),v60,z0,tPen\WObj:=wPaper;
    MoveL Offs(pOrigin,276.46,162.85,0.00),v40,z0,tPen\WObj:=wPaper;
    MoveL Offs(pOrigin,276.69,161.99,0.00),v40,z0,tPen\WObj:=wPaper;
    MoveL Offs(pOrigin,279.54,164.84,0.00),v40,z0,tPen\WObj:=wPaper;
    MoveL Offs(pOrigin,279.11,164.95,0.00),v40,z0,tPen\WObj:=wPaper;
    MoveL Offs(pOrigin,278.05,164.95,0.00),v40,z0,tPen\WObj:=wPaper;
    MoveL Offs(pOrigin,278.26,166.01,0.00),v40,z0,tPen\WObj:=wPaper;
    MoveL Offs(pOrigin,279.32,166.01,0.00),v40,z0,tPen\WObj:=wPaper;
    MoveL Offs(pOrigin,279.54,167.06,0.00),v40,z0,tPen\WObj:=wPaper;
    MoveL Offs(pOrigin,278.48,167.06,0.00),v40,z0,tPen\WObj:=wPaper;
    MoveL Offs(pOrigin,277.75,167.53,0.00),v40,z0,tPen\WObj:=wPaper;
    MoveL Offs(pOrigin,280.76,170.54,0.00),v40,z0,tPen\WObj:=wPaper;
    MoveL Offs(pOrigin,280.18,170.23,0.00),v40,z0,tPen\WObj:=wPaper;
    MoveL Offs(pOrigin,279.11,170.23,0.00),v40,z0,tPen\WObj:=wPaper;
    MoveL Offs(pOrigin,279.32,171.29,0.00),v40,z0,tPen\WObj:=wPaper;
  ENDPROC

